	                         Search window
	                          <--------|
	Data                              PEC
	|----------------------------------|------------------------------------------|
	|                           XXXXXXXX                                          |
	|----------------------------------|------------------------------------------|
	                                   |
	Conveyor                           |
	|----------------------------------|------------------------------------------|
	|                      YYYYYYYY    |                                          |
	|                      YYYYYYYY    |                                          |
	|                      YYYYYYYY    |                                          |
	|----------------------------------|------------------------------------------|
	*)
	(* Data detected without PEC signal.*)
	            IF (#s_R_TRIG_PositiveDataFound.Q
	                AND NOT #sx_ParcelDetected)
	            THEN
	                #si_GINToWrite := 0;
	                // Double data detection loop.
	                FOR #si_i := #si_PositionToUpdate TO #si_PECPosition + (#si_SearchWindow * #si_Direction) BY #si_Direction DO
	                    // Data found in a search window.
	                    IF (#iqa_TrackingData[#si_i] > 0)
	                    THEN
	                        // First GIN found.
	                        IF (#si_GINToWrite = 0)
	                        THEN
	                            // Get the GIN if it's different than last updated GIN.
	                            IF #iqa_TrackingData[#si_i] <> #si_LastUpdatedGIN THEN
	                                #si_GINToWrite := #iqa_TrackingData[#si_i];
	                            END_IF;
	                            // If the first GIN was found, the scan loop conitues to check if there is no other data.
	                        ELSE
	                            // Next found data is different than the first one. Double data detected.
	                            IF (#iqa_TrackingData[#si_i] <> #si_GINToWrite)
	                            THEN
	                                #sx_DoubleDataFound := TRUE;
	                                // First found GIN is marked as a lost one and the GIN is stored in a FIFO register.
	                                IF ("DB_GIN".GIN[#si_GINToWrite].General.Lost = FALSE)
	                                THEN
	                                    "DB_GIN".GIN[#si_GINToWrite].General.Lost := TRUE;

	                                    "FC_Fifo"(ic_Mode := 'W',
	                                              qUDT_Status => #sUDT_LostGINFIFOStatus,
	                                              qx_Error => #sx_LostGINFIFOError,
	                                              qx_Warning => #sx_LostGINFIFOWarning,
	                                              iqv_Data := #si_GINToWrite,
	                                              iqUDT_FifoHeader := #iqUDT_FifoHeader,
	                                              iqv_DataBuffer := #iqa_FifoData);

	                                    // Update statistics
	                                    #ss_LostParcelsCounters.Total += 1;
	                                    #ss_LostParcelsCounters.DoubleData += 1;


	                                    ////////////////////

	                                    IF #si_GINToWrite >= 1000 THEN
	                                        #ss_LostValidParcelsCounters.Total += 1;
	                                        #ss_LostValidParcelsCounters.DoubleData += 1;
	                                    END_IF;

	                                    ////////////////
	                                END_IF;

	                                // Second found GIN is marked as a lost one and the GIN is stored in a FIFO register.
	                                IF ("DB_GIN".GIN[#iqa_TrackingData[#si_i]].General.Lost = FALSE)
	                                THEN
	                                    "DB_GIN".GIN[#iqa_TrackingData[#si_i]].General.Lost := TRUE;

	                                    "FC_Fifo"(ic_Mode := 'W',
	                                              qUDT_Status => #sUDT_LostGINFIFOStatus,
	                                              qx_Error => #sx_LostGINFIFOError,
	                                              qx_Warning => #sx_LostGINFIFOWarning,
	                                              iqv_Data := #iqa_TrackingData[#si_i],
	                                              iqUDT_FifoHeader := #iqUDT_FifoHeader,
	                                              iqv_DataBuffer := #iqa_FifoData);

	                                    // Update statistics
	                                    #ss_LostParcelsCounters.Total += 1;
	                                    #ss_LostParcelsCounters.DoubleData += 1;

	                                    ////////////////////

	                                    IF #iqa_TrackingData[#si_i] >= 1000 THEN
	                                        #ss_LostValidParcelsCounters.Total += 1;
	                                        #ss_LostValidParcelsCounters.DoubleData += 1;
	                                    END_IF;

	                                    ////////////////
	                                    //
	                                END_IF;
	                                // Stop search window scan in case of double data detection
	                                EXIT;
	                            END_IF;
	                        END_IF;
	                    END_IF;
	                END_FOR;

	                // Becasue the data was found as a first one, GIN is stored and the logic to wait for a parcel is enebaled.
	                // If the double data was found there is no need to wait for a parcel. Data has been marked as a lost one.
	                IF NOT #sx_DoubleDataFound
	                THEN
	                    #sx_ParcelWaitEnable := TRUE;
	                END_IF;

	                #sx_DoubleDataFound := FALSE;
	(*
	Data and PEC signal detected at the same time - perfect match

	                         Search window
	                          <--------|
	Data                              PEC
	|----------------------------------|------------------------------------------|
	|                           XXXXXXXX                                          |
	|----------------------------------|------------------------------------------|
	                                   |
	Conveyor                           |
	|----------------------------------|------------------------------------------|
	|                           XXXXXXXX                                          |
	|                           XXXXXXXX                                          |
	|                           XXXXXXXX                                          |
	|----------------------------------|------------------------------------------|

	or PEC signal found without data or with old ones

	                         Search window
	                          <--------|
	Data                              PEC
	|----------------------------------|------------------------------------------|
	|                    XXXXXXXX      |                                          |
	|----------------------------------|------------------------------------------|
	                                   |
	Conveyor                           |
	|----------------------------------|------------------------------------------|
	|                           XXXXXXXX                                          |
	|                           XXXXXXXX                                          |
	|                           XXXXXXXX                                          |
	|----------------------------------|------------------------------------------|
	*)
	(*Data and PEC signal detected at the same time (perfect match) or PEC signal found without data or with old ones.*)
	            ELSIF (#s_R_TRIG_ParcelFound.Q
	                AND (#s_R_TRIG_PositiveDataFound.Q
	                OR (#iqa_TrackingData[#si_PositionToUpdate] = 0
	                OR #iqa_TrackingData[#si_PositionToUpdate] = #si_LastUpdatedGIN)
	                AND NOT #sx_ParcelWaitEnable))
	            THEN
	                // If the PEC is set as a GIN generation point, skip data detection loop and go to GIN generator.
	                IF (#iUDT_PECUpdateConfiguration.GenerationPoint)
	                THEN
	                    #sx_GenerateGIN := TRUE;
	                    // If the the PEC isn't a generation point, data search loop is enabled.
	                ELSE
	                    #si_GINToWrite := 0;

	                    // Double data detection loop.
	                    FOR #si_i := #si_PositionToUpdate TO
	                        (#si_PECPosition + (#si_SearchWindow * #si_Direction)) BY #si_Direction DO

	                        // Data found in a search window.
	                        IF (#iqa_TrackingData[#si_i] > 0)
	                        THEN
	                            // First GIN found.
	                            IF (#si_GINToWrite = 0)
	                            THEN
	                                // Get the GIN if it's different than last updated GIN.
	                                IF #iqa_TrackingData[#si_i] <> #si_LastUpdatedGIN THEN
	                                    #si_GINToWrite := #iqa_TrackingData[#si_i];

	                                    // PEC/Data deviation acquisition
	                                    #"ss_PEC/DataDeviation".Last := DINT_TO_INT(#si_PECPosition - #si_i);
	                                    #"ss_PEC/DataDeviation".GIN := #si_GINToWrite;
	                                    #"ss_PEC/DataDeviation".Sum -= ABS(#"ss_PEC/DataDeviation".Last);
	                                    #"ss_PEC/DataDeviation".Nr += 1;
	                                    IF #"ss_PEC/DataDeviation".Last = 0 THEN
	                                        #"ss_PEC/DataDeviation".Type := 1;
	                                    ELSIF #"ss_PEC/DataDeviation".Last < 0 THEN
	                                        #"ss_PEC/DataDeviation".Type := 2;
	                                    END_IF;

	                                    // Parcel aligned statistics
	                                    IF (ABS(#"ss_PEC/DataDeviation".Last) > ABS(#si_Displacement - 1))
	                                    THEN
	                                        #ss_AlignedParcelsCounters.Total += 1;
	                                        #ss_AlignedParcelsCounters.PECNoData += 1;
	                                    END_IF;
	                                END_IF;
	                                // If the first GIN was found, the scan loop conitues to check if there is no other data.
	                            ELSE
	                                // Next found data is different than the first one. Double data detected.
	                                IF (#iqa_TrackingData[#si_i] <> #si_GINToWrite)
	                                THEN
	                                    // First found GIN is marked as a lost one and the GIN is stored in a FIFO register.
	                                    IF ("DB_GIN".GIN[#si_GINToWrite].General.Lost = FALSE)
	                                    THEN
	                                        "DB_GIN".GIN[#si_GINToWrite].General.Lost := TRUE;
	                                        "FC_Fifo"(ic_Mode := 'W',
	                                                  qUDT_Status => #sUDT_LostGINFIFOStatus,
	                                                  qx_Error => #sx_LostGINFIFOError,
	                                                  qx_Warning => #sx_LostGINFIFOWarning,
	                                                  iqv_Data := #si_GINToWrite,
	                                                  iqUDT_FifoHeader := #iqUDT_FifoHeader,
	                                                  iqv_DataBuffer := #iqa_FifoData);

	                                        // PEC/Data deviation acquisition
	                                        #"ss_PEC/DataDeviation".GIN := #si_GINToWrite;
	                                        #"ss_PEC/DataDeviation".Type := 4;

	                                        // Update statistics
	                                        #ss_LostParcelsCounters.Total += 1;
	                                        #ss_LostParcelsCounters.DoubleData += 1;

	                                        ////////////////////

	                                        IF #si_GINToWrite >= 1000 THEN
	                                            #ss_LostValidParcelsCounters.Total += 1;
	                                            #ss_LostValidParcelsCounters.DoubleData += 1;
	                                        END_IF;

	                                        ////////////////
	                                        //
	                                    END_IF;

	                                    // Second found GIN is marked as a lost one and the GIN is stored in a FIFO register.
	                                    IF ("DB_GIN".GIN[#iqa_TrackingData[#si_i]].General.Lost = FALSE)
	                                    THEN
	                                        "DB_GIN".GIN[#iqa_TrackingData[#si_i]].General.Lost := TRUE;
	                                        "FC_Fifo"(ic_Mode := 'W',
	                                                  qUDT_Status => #sUDT_LostGINFIFOStatus,
	                                                  qx_Error => #sx_LostGINFIFOError,
	                                                  qx_Warning => #sx_LostGINFIFOWarning,
	                                                  iqv_Data := #iqa_TrackingData[#si_i],
	                                                  iqUDT_FifoHeader := #iqUDT_FifoHeader,
	                                                  iqv_DataBuffer := #iqa_FifoData);

	                                        // Update statistics
	                                        #ss_LostParcelsCounters.Total += 1;
	                                        #ss_LostParcelsCounters.DoubleData += 1;

	                                        ////////////////////

	                                        IF #iqa_TrackingData[#si_i] >= 1000 THEN
	                                            #ss_LostValidParcelsCounters.Total += 1;
	                                            #ss_LostValidParcelsCounters.DoubleData += 1;
	                                        END_IF;

	                                        ////////////////
	                                        //
	                                    END_IF;
	                                    // Stop search window scan in case of double data detection
	                                    EXIT;
	                                END_IF;
	                            END_IF;
	                        END_IF;
	                    END_FOR;

	                    // GIN not found in a search window
	                    IF (#si_GINToWrite = 0)
	                    THEN
	                        #sx_GenerateGIN := TRUE;
	                        #si_UnknownParcelsCounters.DataNotFound += 1;
	                    END_IF;

	                    // Found GIN is a lost one - generate unknown GIN
	                    // Found GIN isn't lost or it's negative - don't do anything
	                    IF (#si_GINToWrite > 0)
	                    THEN
	                        IF ("DB_GIN".GIN[#si_GINToWrite].General.Lost)
	                        THEN
	                            #sx_GenerateGIN := TRUE;
	                            #si_UnknownParcelsCounters.LostParcelFound += 1;
	                        END_IF;
	                    END_IF;
	                END_IF;

	                (*Second parcel has been found during data update. Situation can occur when search window is too short
	                  and the data is shifted. In that case found GIN will be marked as a lost one and new unknown GIN will be
	                  generated. Negative GIN will be ignored.*)
	            ELSIF (#s_R_TRIG_ParcelFound.Q
	                AND (#iqa_TrackingData[#si_PositionToUpdate] <> 0
	                AND #iqa_TrackingData[#si_PositionToUpdate] <> #si_LastUpdatedGIN)
	                AND NOT #sx_ParcelWaitEnable)
	            THEN
	                IF (#iqa_TrackingData[#si_PositionToUpdate] > 0)
	                THEN
	                    IF ("DB_GIN".GIN[#iqa_TrackingData[#si_PositionToUpdate]].General.Lost = FALSE)
	                    THEN
	                        "DB_GIN".GIN[#iqa_TrackingData[#si_PositionToUpdate]].General.Lost := TRUE;
	                        "FC_Fifo"(ic_Mode := 'W',
	                                  qUDT_Status => #sUDT_LostGINFIFOStatus,
	                                  qx_Error => #sx_LostGINFIFOError,
	                                  qx_Warning => #sx_LostGINFIFOWarning,
	                                  iqv_Data := #iqa_TrackingData[#si_PositionToUpdate],
	                                  iqUDT_FifoHeader := #iqUDT_FifoHeader,
	                                  iqv_DataBuffer := #iqa_FifoData);

	                        // Update statistics
	                        #ss_LostParcelsCounters.Total += 1;
	                        #ss_LostParcelsCounters.DoubleData += 1;

	                        ////////////////////

	                        IF #iqa_TrackingData[#si_PositionToUpdate] >= 1000 THEN
	                            #ss_LostValidParcelsCounters.Total += 1;
	                            #ss_LostValidParcelsCounters.DoubleData += 1;
	                        END_IF;

	                        ////////////////
	                        //
	                    END_IF;
	                END_IF;

	                // Generate GIN
	                #sx_GenerateGIN := TRUE;
	                #si_UnknownParcelsCounters.LostParcelFound += 1;

	                (*Second data has been found during data update. Situation can occur when search window is too short
	                  and the data is shifted. In that case found GIN will be marked as a lost one.*)
	            ELSIF (#s_R_TRIG_PositiveDataFound.Q
	                AND #sx_ParcelDetected
	                AND #iqa_TrackingData[#si_PositionToUpdate] <> #si_GINToWrite)
	            THEN
	                // Mark GIN as a lost one
	                IF ("DB_GIN".GIN[#iqa_TrackingData[#si_PositionToUpdate]].General.Lost = FALSE)
	                THEN
	                    "DB_GIN".GIN[#iqa_TrackingData[#si_PositionToUpdate]].General.Lost := TRUE;
	                    "FC_Fifo"(ic_Mode := 'W',
	                              qUDT_Status => #sUDT_LostGINFIFOStatus,
	                              qx_Error => #sx_LostGINFIFOError,
	                              qx_Warning => #sx_LostGINFIFOWarning,
	                              iqv_Data := #iqa_TrackingData[#si_PositionToUpdate],
	                              iqUDT_FifoHeader := #iqUDT_FifoHeader,
	                              iqv_DataBuffer := #iqa_FifoData);

	                    // Update statistics
	                    #ss_LostParcelsCounters.Total += 1;
	                    #ss_LostParcelsCounters.DoubleData += 1;

	                    ////////////////////

	                    IF #iqa_TrackingData[#si_PositionToUpdate] >= 1000 THEN
	                        #ss_LostValidParcelsCounters.Total += 1;
	                        #ss_LostValidParcelsCounters.DoubleData += 1;
	                    END_IF;

	                    ////////////////
	                END_IF;
	            END_IF;

	        END_REGION

	        REGION 10.5 – GIN generator

	            (*Used to generate new GIN. If the PEC position is a generation point, the number is taken from an internal GIN range.
	              If it's not, then GIN is taken from a global unknown GIN range.*)

	            IF (#sx_GenerateGIN)
	            THEN
	                // Generation point.
	                IF (#iUDT_PECUpdateConfiguration.GenerationPoint)
	                THEN
	                    // Generate GIN from a valid GIN range.
	                    IF (#ss_ValidGINRange.GIN <= #ss_ValidGINRange.End)
	                    THEN
	                        #si_GINToWrite := #ss_ValidGINRange.GIN;
	                        #ss_ValidGINRange.GIN += 1;
	                    ELSE
	                        #si_GINToWrite := #ss_ValidGINRange.Start;
	                        #ss_ValidGINRange.GIN := #ss_ValidGINRange.Start + 1;
	                    END_IF;
	                    // Unknown GIN generator.
	                ELSE
	                    // Generate GIN from a unknown GIN range.
	                    IF (#iqUDT_UnknownGINRange.GIN <= #iqUDT_UnknownGINRange.End)
	                    THEN
	                        #si_GINToWrite := #iqUDT_UnknownGINRange.GIN;
	                        #iqUDT_UnknownGINRange.GIN += 1;
	                    ELSE
	                        #si_GINToWrite := #iqUDT_UnknownGINRange.Start;
	                        #iqUDT_UnknownGINRange.GIN := #iqUDT_UnknownGINRange.Start + 1;
	                    END_IF;

	                    // Unknwn parcels statistics.
	                    #si_UnknownParcelsCounters.Total += 1;
	                END_IF;

	                // Reset generte GIN command.
	                #sx_GenerateGIN := FALSE;

	                // GIN record is cleared with configured default GIN record while it's generated.
	                "DB_GIN".GIN[#si_GINToWrite] := "DB_GINDefault".GIN[#iUDT_PECUpdateConfiguration.DefaultGIN];
	            END_IF;

	            #qi_GINwrite := #si_GINToWrite;

	        END_REGION


	        REGION 10.6 – PEC position data update

	            (*While parcel is detected, calculated GIN is written into the PEC position record.
	              If not, then the record is cleared with 0. Negative GIN is ignored or deleted, depending on configuration.*)

	            IF (#sx_ParcelDetected)
	            THEN

	                "FC_WriteGIN"(ii_GIN := #si_GINToWrite,
	                              ii_PositionToWrite := #si_PositionToUpdate,
	                              ii_NumberOfPositions := 1,
	                              ix_Direction := TRUE,
	                              iqa_TrackingData := #iqa_TrackingData);

	            ELSE
	                IF (#iqa_TrackingData[#si_PositionToUpdate] > 0
	                    OR #iUDT_PECUpdateConfiguration.NegativeGINDelete)
	                THEN

	                    "FC_WriteGIN"(ii_GIN := #ci_ZeroGIN,
	                                  ii_PositionToWrite := #si_PositionToUpdate,
	                                  ii_NumberOfPositions := 1,
	                                  ix_Direction := TRUE,
	                                  iqa_TrackingData := #iqa_TrackingData);

	                END_IF;
	            END_IF;

	        END_REGION

	        REGION 10.7 – Parcel waiting logic

	            (*Parcel waiting logic is used to wait for the photoeye signal for a search window distance.*)
	            IF (#sx_ParcelWaitEnable)
	            THEN
	                // Counting parcel wait distance depending on conveyor running direction if not detected.
	                IF (NOT #sx_ParcelDetected)
	                THEN
	                    IF (#si_Direction = 1)
	                    THEN
	                        #si_ParcelWaitDistance += 1;

	                    ELSE
	                        #si_ParcelWaitDistance -= ABS(#si_Displacement);   //1;
	                    END_IF;

	                    // Parcel detected - stop waiting, use found GIN to update.
	                ELSE
	                    // PEC/Data deviation acquisition
	                    #"ss_PEC/DataDeviation".Type := 3;
	                    #"ss_PEC/DataDeviation".Last := #si_ParcelWaitDistance;
	                    #"ss_PEC/DataDeviation".GIN := #si_GINToWrite;
	                    #"ss_PEC/DataDeviation".Sum += ABS(#"ss_PEC/DataDeviation".Last);
	                    #"ss_PEC/DataDeviation".Nr += 1;


	                    // Parcel aligned statistics
	                    IF (#"ss_PEC/DataDeviation".Last > ABS(#si_Displacement - 1))
	                    THEN
	                        #ss_AlignedParcelsCounters.Total += 1;
	                        #ss_AlignedParcelsCounters.DataNoPEC += 1;
	                    END_IF;

	                    // Parcel waiting logic reset.
	                    #sx_ParcelWaitEnable := FALSE;
	                    #si_ParcelWaitDistance := 0;
	                END_IF;
	            END_IF;

	            // Parcel not found in a search window - stop waiting, mark found GIN as a lost one.
	            IF (ABS(#si_ParcelWaitDistance) = #si_SearchWindow)
	                AND (#si_GINToWrite > 0)
	            THEN
	                // Parcel lost
	                IF "DB_GIN".GIN[#si_GINToWrite].General.Lost = FALSE THEN
	                    "DB_GIN".GIN[#si_GINToWrite].General.Lost := TRUE;
	                    "FC_Fifo"(ic_Mode := 'W',
	                              qUDT_Status => #sUDT_LostGINFIFOStatus,
	                              qx_Error => #sx_LostGINFIFOError,
	                              qx_Warning => #sx_LostGINFIFOWarning,
	                              iqv_Data := #si_GINToWrite,
	                              iqUDT_FifoHeader := #iqUDT_FifoHeader,
	                              iqv_DataBuffer := #iqa_FifoData);

	                    // PEC/Data deviation acquisition
	                    #"ss_PEC/DataDeviation".Type := 5;
	                    #"ss_PEC/DataDeviation".Last := #si_ParcelWaitDistance;
	                    #"ss_PEC/DataDeviation".GIN := #si_GINToWrite;
	                    #"ss_PEC/DataDeviation".Sum += ABS(#"ss_PEC/DataDeviation".Last);
	                    #"ss_PEC/DataDeviation".Nr += 1;

	                    // Parcel waiting logic reset.
	                    #si_ParcelWaitDistance := 0;
	                    #sx_ParcelWaitEnable := FALSE;

	                    // Lost parcels ina  row counter.
	                    #si_LostParcelsInARow += 1;

	                    // Update statistics.
	                    #ss_LostParcelsCounters.Total += 1;
	                    #ss_LostParcelsCounters.ParcelNotFound += 1;

	                    ////////////////////

	                    IF #si_GINToWrite >= 1000 THEN
	                        #ss_LostValidParcelsCounters.Total += 1;
	                        #ss_LostValidParcelsCounters.ParcelNotFound += 1;
	                    END_IF;

	                    ////////////////
	                    //
	                END_IF;

	            END_IF;

	            // Reset monitoring in case of going backwards.
	            IF (#si_ParcelWaitDistance = 0
	                AND NOT #sx_ParcelDetected
	                AND #sx_InvalidDirection)
	            THEN
	                #sx_ParcelWaitEnable := FALSE;
	            END_IF;

	            #sx_InvalidDirection := ((#si_Direction = 1
	            AND #si_ParcelWaitDistance < 0)
	            OR (#si_Direction = -1
	            AND #si_ParcelWaitDistance > 0));

	        END_REGION

	        REGION 10.8 – Last updated GIN

	            (*Last updated GIN to avoid processing the same data.*)
	            IF (#s_R_TRIG_DataFound.Q)
	            THEN
	                #si_LastUpdatedGIN := #iqa_TrackingData[#si_PositionToUpdate];
	            END_IF;

	        END_REGION

	        REGION 10.8 – Update displacement

	            #si_Displacement := #si_Displacement - #si_Direction;

	        END_REGION

	    END_WHILE;

	END_REGION

	REGION 11 – Length measurement



	    (*Length and gap measurements can be enabled via PEC update configuration*)
	    #sFB_LengthMeasurement(ii_PECPosition := #si_PECPosition,
	                           ii_Displacement := #iqUDT_ConveyorInterface.Displacement,
	                           ix_LengthMeasurementEnable := #iUDT_PECUpdateConfiguration.ParcelLengthMeasurement OR #sx_LengthMeasurementEnable,
	                           ix_GapMeasurementEnable := #iUDT_PECUpdateConfiguration.GapLengthMeasurement,
	                           iqa_TrackingData := #iqa_TrackingData);

	    IF #iqa_TrackingData[#si_PECPosition] > 0
	        AND #iqa_TrackingData[#si_PECPosition] >= #iqUDT_UnknownGINRange.Start
	        AND #iqa_TrackingData[#si_PECPosition] <= #iqUDT_UnknownGINRange.End
	    THEN

	        #sx_LengthMeasurementEnable := "DB_GIN".GIN[#iqa_TrackingData[#si_PECPosition]].General.Length = 0;
	    ELSE

	        #sx_LengthMeasurementEnable := FALSE;

	    END_IF;

	END_REGION

	REGION 12 – Teaching done

	    // Average slip calculation
	    #si_AverageSlip := #"ss_PEC/DataDeviation".Sum / #"ss_PEC/DataDeviation".Nr;
	    #si_CalculatedLengthCorrection := DINT_TO_INT(#iUDT_ConveyorCommonConfiguration.LengthCorrection) + #si_AverageSlip * 10;
	    IF (#sx_TeachingMode                                                                                                            // Teaching mode enabled
	        AND #si_NumberOfTeachedParcels = #iUDT_PECUpdateConfiguration.NrOfTeachParcels)                                                 // Number of teaching parcels equal to the preset one                                                                                                                                                              // Teaching mode enabled ("sx_TeachMode")
	    THEN

	        #si_CalculatedLengthCorrection := DINT_TO_INT(#iUDT_ConveyorCommonConfiguration.LengthCorrection) + #si_AverageSlip * 10;
	        #sx_TeachingMode := FALSE;
	        #si_NumberOfTeachedParcels := 0;

	    END_IF;

	END_REGION

	REGION 13 – Performance

	    (*Performnce is a percentage ratio between number of lost parcels and total number of data, used to monitor data update efficiency.*)

	    IF (#sdi_TotalNumberOfData >= #ss_LostParcelsCounters.Total
	        AND #sdi_TotalNumberOfData > 0)
	    THEN
	        #slr_Performance := 100.0 - INT_TO_LREAL(#ss_LostParcelsCounters.Total) / #sdi_TotalNumberOfData * 100.0;
	    END_IF;

	    // Warning is generated if performance drops below 80%.
	    #qUDT_Status.LowPerformance := #slr_Performance < 80;

	END_REGION

	REGION 14 – Reset statistics

	    // Statistics are reset if reset signal is given.
	    IF #iqUDT_ConveyorInterface.ResetStatistics
	    THEN
	        #sdi_TotalNumberOfParcels := 0;
	        #ss_AlignedParcelsCounters.Total := 0;
	        #ss_AlignedParcelsCounters.PECNoData := 0;
	        #ss_AlignedParcelsCounters.DataNoPEC := 0;
	        #ss_LostParcelsCounters.Total := 0;
	        #ss_LostParcelsCounters.DoubleData := 0;
	        #ss_LostParcelsCounters.ParcelNotFound := 0;
	        #ss_LostValidParcelsCounters.Total := 0;
	        #ss_LostValidParcelsCounters.DoubleData := 0;
	        #ss_LostValidParcelsCounters.ParcelNotFound := 0;
	        #sdi_TotalNumberOfData := 0;
	        #si_UnknownParcelsCounters.Total := 0;
	        #si_UnknownParcelsCounters.LostParcelFound := 0;
	        #si_UnknownParcelsCounters.DataNotFound := 0;
	        #"ss_PEC/DataDeviation".Sum := 0;
	        #"ss_PEC/DataDeviation".Nr := 0;
	        #slr_Performance := 100;

	    END_IF;

	END_REGION

	REGION 15 – Too many lost parcels error

	    (*Error is generated if too many parcels will is marked as a lost one in a row*)
	    IF (#si_LostParcelsInARow >= #iUDT_PECUpdateConfiguration.MaxLost)
	    THEN
	        #qUDT_Status.TooManyLost := TRUE;
	    END_IF;

	END_REGION

	REGION 16 – Statistics

	    // Too many lost
	    #s_R_TRIG_TooManyLost(CLK := #qUDT_Status.TooManyLost);
	    IF #qUDT_Status.TooManyLost
	        OR #iqUDT_ConveyorInterface.ResetStatistics
	    THEN
	        "FC_Statistics"(ix_Reset := #iqUDT_ConveyorInterface.ResetStatistics,
	                        ix_Activate := #qUDT_Status.TooManyLost,
	                        ix_RTrigActivate := #s_R_TRIG_TooManyLost.Q,
	                        iqUDT_Statistics := #iqUDT_Statistics.TooManyLost);
	    END_IF;

	    // Total number of parcels
	    #iqUDT_Statistics.TotalNrOfParcels := #sdi_TotalNumberOfParcels;

	END_REGION

	REGION 17 – Internal tracking warning and error

	    // Internal tracking warning
	    IF (#qUDT_Status.LowPerformance
	        OR #sx_LostGINFIFOWarning)
	    THEN
	        #iqUDT_ConveyorInterface.InternalWarningTracking := TRUE;
	    END_IF;

	    // Internal tracking error
	    IF #qUDT_Status.TooManyLost
	    THEN
	        #iqUDT_ConveyorInterface.InternalErrorTracking := TRUE;
	    END_IF;

	    // Configuration error
	    IF (#sx_InvalidDisplacement
	        OR #sx_InvalidGINRange
	        OR #sx_InvalidSearchWindow)
	    THEN
	        #iqUDT_ConveyorInterface.ConfigurationError := TRUE;
	    END_IF;

	END_REGION
END_FUNCTION_BLOCK

FUNCTION_BLOCK "FB_CaljanV2"
TITLE = FB_Unloader
{ S7_Optimized_Access := 'TRUE' }
AUTHOR : MHSE
FAMILY : Equimpent
VERSION : 1.2
// ATTRIBUTES
// AUTO_NUMBER = True
// BLOCK_NUMBER = 201
// END_ATTRIBUTES
//Function block to control unloader.
   VAR_INPUT
      iUDT_CaljanConfiguration { ExternalAccessible := 'False'; ExternalVisible := 'False'; ExternalWritable := 'False'} : "UDT_CaljanConfigurationV2";   // Caljan configuration structure
      iUDT_CaljanReceive { ExternalAccessible := 'False'; ExternalVisible := 'False'; ExternalWritable := 'False'} : "UDT_CaljanReceiveV2";   // Caljan receive structure
      ix_SafetyReset { ExternalAccessible := 'False'; ExternalVisible := 'False'; ExternalWritable := 'False'} : Bool;   // Safety reset
      ix_SafetyOk { ExternalAccessible := 'False'; ExternalVisible := 'False'; ExternalWritable := 'False'} : Bool;   // TRUE when Safety Circuit of the Conveyor is healthy
      ix_24vOk { ExternalAccessible := 'False'; ExternalVisible := 'False'; ExternalWritable := 'False'} : Bool;   // TRUE when 24VDC is healthy
      ix_400vOk { ExternalAccessible := 'False'; ExternalVisible := 'False'; ExternalWritable := 'False'} : Bool;   // TRUE when 400VAC is healthy
      ix_HardwareOK { ExternalAccessible := 'False'; ExternalVisible := 'False'; ExternalWritable := 'False'} : Bool;   // TRUE when the PN node(s) are ok
      ix_ExternalRequestDieBack { ExternalAccessible := 'False'; ExternalVisible := 'False'; ExternalWritable := 'False'} : Bool;   // External request die back
      ix_ExternalRequestHold { ExternalAccessible := 'False'; ExternalVisible := 'False'; ExternalWritable := 'False'} : Bool;   // External request hold
      ix_ExternalRunReverse { ExternalAccessible := 'False'; ExternalVisible := 'False'; ExternalWritable := 'False'} : Bool;   // External request only for unloder mode - TRUE when conveyor should run in reverse direction
      ix_ResetEnergySave { ExternalAccessible := 'False'; ExternalVisible := 'False'; ExternalWritable := 'False'} : Bool;   // Reset energy save mode timer
      ix_SimulationModeActive { ExternalAccessible := 'False'; ExternalVisible := 'False'; ExternalWritable := 'False'} : Bool;   // TRUE when simulation mode is active
      ix_CaljanMode { ExternalAccessible := 'False'; ExternalVisible := 'False'; ExternalWritable := 'False'} : Int;   // Choosing device 1=loader, 2=unloader
      ix_BufferPEC { ExternalAccessible := 'False'; ExternalVisible := 'False'; ExternalWritable := 'False'} : Bool;   // Buufer PEC
   END_VAR

   VAR_OUTPUT
      qUDT_HMIStatus { ExternalAccessible := 'False'; ExternalVisible := 'False'; ExternalWritable := 'False'} : "UDT_CaljanStatusV2";   // HMI status structure
      qUDT_Status { ExternalAccessible := 'False'; ExternalVisible := 'False'; ExternalWritable := 'False'} : "UDT_CommonStatus";   // Common status structure
      qUDT_CaljanSend { ExternalAccessible := 'False'; ExternalVisible := 'False'; ExternalWritable := 'False'} : "UDT_CaljanSendV2";   // Caljan send structure
   END_VAR

   VAR_IN_OUT
      iqUDT_EquipmentControl : "UDT_EquipmentControl";   // Equipment control structure
      iqUDT_CaljanCommand : "UDT_CaljanCommand";   // Caljan HMI control
      iqUDT_ConveyorInterface : "UDT_ConveyorInterface";   // Interface structure
      iqUDT_HandShake : "UDT_ConveyorHandshake";   // Handshake structure
      iqUDT_HandShakeUp : "UDT_ConveyorHandshake";   // Upstream handshake structure
      iqUDT_Statistics : "UDT_CaljanStatisticsV2";   // Statistics structure
   END_VAR

   VAR
      s_FB_ResetPulseTimer { ExternalAccessible := 'False'; ExternalVisible := 'False'; ExternalWritable := 'False'; S7_SetPoint := 'False'} : "FB_TimerOnOffDelay";   // Timer on/off delay for reset pulse
      s_FB_CascadeModeTimer { ExternalAccessible := 'False'; ExternalVisible := 'False'; ExternalWritable := 'False'; S7_SetPoint := 'False'} : "FB_TimerOnOffDelay";   // Timer on/off delay for cascade mode
      s_FB_TimerOnOffDelayCheck24V { ExternalAccessible := 'False'; ExternalVisible := 'False'; ExternalWritable := 'False'; S7_SetPoint := 'False'} : "FB_TimerOnOffDelay";   // Timer on/off delay to allow startup before fault is generated
      s_FB_TimerOnOffDelayCheck400V { ExternalAccessible := 'False'; ExternalVisible := 'False'; ExternalWritable := 'False'; S7_SetPoint := 'False'} : "FB_TimerOnOffDelay";   // Timer on/off delay to allow startup before fault is generated
      s_UDT_CommonStatus { ExternalAccessible := 'False'; ExternalVisible := 'False'; ExternalWritable := 'False'; S7_SetPoint := 'False'} : "UDT_CommonStatus";   // Common status structure
      s_UDT_CommonStatusOld { ExternalAccessible := 'False'; ExternalVisible := 'False'; ExternalWritable := 'False'; S7_SetPoint := 'False'} : "UDT_CommonStatus";   // Auxiliary status structure
      s_UDT_HMIStatus { ExternalAccessible := 'False'; ExternalVisible := 'False'; ExternalWritable := 'False'; S7_SetPoint := 'False'} : "UDT_CaljanStatusV2";   // HMI status structure
      s_UDT_PNDevice { ExternalAccessible := 'False'; ExternalVisible := 'False'; ExternalWritable := 'False'; S7_SetPoint := 'False'} : "UDT_PNDevice";   // PN device info structure
      sa_PNPortsStatus { ExternalAccessible := 'False'; ExternalVisible := 'False'; ExternalWritable := 'False'} : Array[1..8] of Bool;   // TRUE when specific port has an error
      R_TRIG_EnergySave {InstructionName := 'R_TRIG'; LibVersion := '1.0'; ExternalAccessible := 'False'; ExternalVisible := 'False'; ExternalWritable := 'False'; S7_SetPoint := 'False'} : R_TRIG;   // Rising edge for energy save
      R_TRIG_ConveyorUp {InstructionName := 'R_TRIG'; LibVersion := '1.0'; ExternalAccessible := 'False'; ExternalVisible := 'False'; ExternalWritable := 'False'; S7_SetPoint := 'False'} : R_TRIG;   // Rising edge of automatic active
      R_TRIG_ConveyorDown {InstructionName := 'R_TRIG'; LibVersion := '1.0'; ExternalAccessible := 'False'; ExternalVisible := 'False'; ExternalWritable := 'False'; S7_SetPoint := 'False'} : R_TRIG;   // Rising edge of automatic not active
      R_TRIG_NotHealthy {InstructionName := 'R_TRIG'; LibVersion := '1.0'; ExternalAccessible := 'False'; ExternalVisible := 'False'; ExternalWritable := 'False'; S7_SetPoint := 'False'} : R_TRIG;   // Rising edge trigger if extendable not healthy
      R_TRIG_SafetyOk {InstructionName := 'R_TRIG'; LibVersion := '1.0'; ExternalAccessible := 'False'; ExternalVisible := 'False'; ExternalWritable := 'False'; S7_SetPoint := 'False'} : R_TRIG;   // Rising edge trigger safety is ok
      s_R_TRIG_PNSlaveError {InstructionName := 'R_TRIG'; LibVersion := '1.0'; ExternalAccessible := 'False'; ExternalVisible := 'False'; ExternalWritable := 'False'; S7_SetPoint := 'False'} : R_TRIG;   // Rising edge for PN error
      s_R_TRIG_PNSlaveNotOnline {InstructionName := 'R_TRIG'; LibVersion := '1.0'; ExternalAccessible := 'False'; ExternalVisible := 'False'; ExternalWritable := 'False'; S7_SetPoint := 'False'} : R_TRIG;   // Rising edge for PN not online
      s_R_TRIG_ResetEnergySaveRunMode {InstructionName := 'R_TRIG'; LibVersion := '1.0'; ExternalAccessible := 'False'; ExternalVisible := 'False'; ExternalWritable := 'False'; S7_SetPoint := 'False'} : R_TRIG;   // Rising edge trigger reset energy save mode
      s_R_TRIG_ResetEnergySaveBufferMode {InstructionName := 'R_TRIG'; LibVersion := '1.0'; ExternalAccessible := 'False'; ExternalVisible := 'False'; ExternalWritable := 'False'; S7_SetPoint := 'False'} : R_TRIG;   // Rising edge trigger reset energy save mode
      s_R_TRIG_ResetEnergySaveActive {InstructionName := 'R_TRIG'; LibVersion := '1.0'; ExternalAccessible := 'False'; ExternalVisible := 'False'; ExternalWritable := 'False'; S7_SetPoint := 'False'} : R_TRIG;   // Rising edge trigger reset energy save mode
   END_VAR
   VAR RETAIN
      sdi_EnergySave { ExternalAccessible := 'False'; ExternalVisible := 'False'; ExternalWritable := 'False'} : DInt;   // Energy save displacement
   END_VAR
   VAR
      sx_Disabled { ExternalAccessible := 'False'; ExternalVisible := 'False'; ExternalWritable := 'False'} : Bool;   // Operation is enabled
      sx_Ready { ExternalAccessible := 'False'; ExternalVisible := 'False'; ExternalWritable := 'False'} : Bool;   // Conveyor Ready to operate in Forward mode
      sx_EnergySaveActive { ExternalAccessible := 'False'; ExternalVisible := 'False'; ExternalWritable := 'False'} : Bool;   // Active energy save mode
      sx_AutomaticActive { ExternalAccessible := 'False'; ExternalVisible := 'False'; ExternalWritable := 'False'} : Bool;   // Forward active
      sx_CascadeStartUp { ExternalAccessible := 'False'; ExternalVisible := 'False'; ExternalWritable := 'False'} : Bool;   // Cascade startup auxiliary bit
      sx_24VOk { ExternalAccessible := 'False'; ExternalVisible := 'False'; ExternalWritable := 'False'} : Bool;   // 24V ok
      sx_400VOk { ExternalAccessible := 'False'; ExternalVisible := 'False'; ExternalWritable := 'False'} : Bool;   // 400V ok
   END_VAR

   VAR CONSTANT
      ci_NumberOfProfinetPorts : Int := 2;   // Number of Profinet ports in device
      ci_PowerSupplyDelayTime : UInt := 4000;   // Power supply delay time
   END_VAR


BEGIN
	(*
	----------------------------------------------------------------------------------------
	|                                                                                      |
	|  Copyright  2023             FORTNA Europe BV                                        |
	|  All Rights Reserved         Netherlands                                             |
	|                                                                                      |
	----------------------------------------------------------------------------------------

	Version history:
	Date        | Version   | Author       | Remark
	----------------------------------------------------------------------------------------
	07/03/2023  | 1.0       | S. Nikodem   | Release TIA 17 | DHL Munich 2023
	20/12/2023  | 1.1       | M. Diebel    | Update
	20/12/2023  | 1.2       | L.Klar       | Energy save mode added
	05/02/20234 | 1.3       | P.Gryszczyk  | Added HardwareOk to Profinet faults reset
	05/02/20234 | 1.4       | L.Klar       | Added dieback condition to unload function
	07/02/20234 | 1.5       | L.Klar       | Buffer mode corrected
	09/02/2024  | 1.6       | P.Gryszczyk  | Changed logic for BufferPEC when using Caljan sensor
	*)

	REGION 1 - Get Device Profinet information

	    "FC_GetDevicePN"(is_PNDeviceName := #iUDT_CaljanConfiguration.PNDeviceName,
	                     ix_SimulationModeActive := #ix_SimulationModeActive,
	                     iqUDT_PND := #s_UDT_PNDevice);

	    "FC_GetPNPortStatus"(ii_NumberOfPorts := #ci_NumberOfProfinetPorts,
	                         iUDT_DevicePNInfo := #s_UDT_PNDevice,
	                         qa_PortFault => #sa_PNPortsStatus);

	END_REGION

	REGION 2 - Initial

	    REGION 2.1 - First PLC cycle

	        IF "DB_Memory".FirstScan
	        THEN
	            #sx_AutomaticActive := FALSE;
	            #iqUDT_HandShakeUp.RTR := FALSE;
	            #iqUDT_HandShakeUp.CascadeStartUp := FALSE;
	            #sx_Disabled := FALSE;
	        END_IF;

	    END_REGION

	    REGION 2.2 - Triggers

	        // Rising edge trigger energy save
	        #R_TRIG_EnergySave(CLK := #s_UDT_CommonStatus.EnergySave);

	        // Rising edge extendable up
	        #R_TRIG_ConveyorUp(CLK := #sx_AutomaticActive AND #sx_Ready);

	        // Rising edge extendable down
	        #R_TRIG_ConveyorDown(CLK := #sx_AutomaticActive AND NOT #sx_Ready);

	        // Rising edge extendable not healthy
	        #R_TRIG_NotHealthy(CLK := #s_UDT_HMIStatus.Specific.NotHealthy);

	        // Rising edge for Profinet error
	        #s_R_TRIG_PNSlaveError(CLK := #s_UDT_HMIStatus.Specific.PNSlaveError);

	        // Rising edge for Profinet not online
	        #s_R_TRIG_PNSlaveNotOnline(CLK := #s_UDT_HMIStatus.Specific.PNSlaveNotOnline);

	        // Rising edge for reset energy save mode

	        #s_R_TRIG_ResetEnergySaveRunMode(CLK := #iUDT_CaljanReceive.RunModeActivated);
	        #s_R_TRIG_ResetEnergySaveBufferMode(CLK := #iUDT_CaljanReceive.StoreModeActivated);
	        #s_R_TRIG_ResetEnergySaveActive(CLK := #sx_EnergySaveActive);


	    END_REGION

	    REGION 2.3 - HMI button Disable operation

	        // Copy HMI command to static memory
	        #sx_Disabled := #iqUDT_CaljanCommand.Disable;

	        // Copy status to HMI
	        #s_UDT_HMIStatus.Specific.Disabled := #sx_Disabled;

	    END_REGION

	    REGION 2.6 - Timers

	        // Hardware will only be available after the delay, so the device has time for the initialisation
	        #s_FB_TimerOnOffDelayCheck24V(iudi_OnDelayTime := #ci_PowerSupplyDelayTime,
	                                      ix_SignalToDelay := #ix_24vOk,
	                                      qx_DelayedSignal => #sx_24VOk);

	        #s_FB_TimerOnOffDelayCheck400V(iudi_OnDelayTime := #ci_PowerSupplyDelayTime,
	                                       ix_SignalToDelay := #ix_400vOk,
	                                       qx_DelayedSignal => #sx_400VOk);

	    END_REGION

	END_REGION

	REGION 3 - Reset Profinet errors

	    IF #iqUDT_EquipmentControl.Command.Reset OR (NOT #ix_HardwareOK AND #s_UDT_HMIStatus.Specific.PNSlaveNotOnline) THEN

	        #s_UDT_HMIStatus.Specific.PNSlaveNotOnline := FALSE;
	        #s_UDT_HMIStatus.Specific.PNSlaveError := FALSE;
	        #s_UDT_HMIStatus.Specific.PNSlaveWarning := FALSE;
	    END_IF;

	END_REGION

	REGION 4 - Errors

	    // Check if PN device is online
	    IF NOT "DB_ProfinetDiagnostic".ProfinetNetworks[#s_UDT_PNDevice.PNNetworknumber].DeviceStatus[#s_UDT_PNDevice.PNDeviceNumber].DeviceState.Exist
	        AND NOT #ix_SimulationModeActive
	        AND #sx_24VOk
	        AND #ix_HardwareOK
	    THEN
	        #s_UDT_HMIStatus.Specific.PNSlaveNotOnline := TRUE;

	    END_IF;

	    // Check if PN ports are healthy
	    IF #sa_PNPortsStatus[1] XOR #sa_PNPortsStatus[2] THEN
	        #s_UDT_HMIStatus.Specific.PNSlaveWarning := TRUE;
	    END_IF;

	    // Check if PN device has an error
	    IF "DB_ProfinetDiagnostic".ProfinetNetworks[#s_UDT_PNDevice.PNNetworknumber].DeviceStatus[#s_UDT_PNDevice.PNDeviceNumber].DeviceState.Error
	        AND NOT #ix_SimulationModeActive
	        AND #sx_24VOk
	        AND NOT #s_UDT_HMIStatus.Specific.PNSlaveWarning
	        AND #ix_HardwareOK
	    THEN
	        #s_UDT_HMIStatus.Specific.PNSlaveError := TRUE;
	    END_IF;

	    // Not healthy
	    #s_UDT_HMIStatus.Specific.NotHealthy := NOT #iUDT_CaljanReceive.Healthy
	    AND #sx_400VOk
	    AND #sx_24VOk
	    AND #ix_HardwareOK
	    AND #ix_SafetyOk;

	    // Common Error
	    #s_UDT_CommonStatus.Error := NOT #sx_24VOk
	    OR NOT #sx_400VOk
	    OR NOT #ix_HardwareOK
	    OR NOT #ix_SafetyOk
	    OR #s_UDT_HMIStatus.Specific.PEC_EoS.Jam
	    OR #s_UDT_HMIStatus.Specific.NotHealthy;


	END_REGION

	REGION 5 - Speed

	    #iqUDT_ConveyorInterface.ActualSpeed := #iUDT_CaljanReceive.ActualSpeed;

	END_REGION

	REGION 6 - Check conditions to set caljan ready

	    #sx_Ready := NOT #s_UDT_CommonStatus.Error;

	END_REGION

	REGION 7 - Stop caljan

	    IF NOT #iqUDT_EquipmentControl.Command.AutomaticOn
	        OR #s_UDT_CommonStatus.Error
	    THEN
	        #sx_AutomaticActive := FALSE;
	        #qUDT_CaljanSend.AllowLoading := FALSE;
	        #qUDT_CaljanSend.AllowUnloading := FALSE;
	        #iqUDT_HandShakeUp.RTR := FALSE;
	        #iqUDT_HandShakeUp.CascadeStartUp := FALSE;
	    END_IF;

	END_REGION

	REGION 8 - Start automatic mode

	    // If start (one shot) is received from system, this is memorised until started in cascade. Later the unloader is started
	    IF #iqUDT_EquipmentControl.Command.Start
	        AND #sx_Ready
	    THEN
	        #sx_AutomaticActive := TRUE;
	    END_IF;

	    //Timer to cascade mode
	    #s_FB_CascadeModeTimer(iudi_OnDelayTime := #iUDT_CaljanConfiguration.CascadeTimeOnDelay,
	                           ix_SignalToDelay := #sx_AutomaticActive,
	                           ix_Enable := #sx_Ready,
	                           qx_DelayedSignal => #sx_CascadeStartUp);

	    #iqUDT_HandShakeUp.CascadeStartUp := #sx_CascadeStartUp;

	    //Automatic mode active
	    #qUDT_CaljanSend.Enable := #sx_AutomaticActive AND NOT #s_R_TRIG_ResetEnergySaveActive.Q;

	END_REGION

	REGION 9 - Automatic mode active

	    REGION 9.1 - Operation

	        (* *******LOADER ******** *)
	        IF #ix_CaljanMode = 1 THEN

	            // Release loading
	            #qUDT_CaljanSend.AllowLoading := #sx_AutomaticActive
	            AND #sx_Ready
	            AND NOT #sx_Disabled
	            AND NOT #ix_ExternalRequestHold
	            AND NOT #sx_EnergySaveActive
	            AND (#iUDT_CaljanReceive.RunModeActivated OR #iUDT_CaljanReceive.StoreModeActivated);

	            #iqUDT_HandShakeUp.RTR := #qUDT_CaljanSend.AllowLoading AND ABS(#iUDT_CaljanReceive.ActualSpeed) > 400;

	        END_IF;

	        (* *******UNLOADER ******** *)
	        IF #ix_CaljanMode = 2
	        THEN

	            // Release unloading
	            #qUDT_CaljanSend.AllowUnloading := #sx_AutomaticActive
	            AND #sx_Ready
	            AND (#iqUDT_HandShake.RTR OR #iUDT_CaljanReceive.PECUnloader)
	            AND NOT #sx_Disabled
	            AND NOT #ix_ExternalRequestHold
	            AND NOT #sx_EnergySaveActive
	            AND NOT #ix_ExternalRunReverse;

	        END_IF;

	    END_REGION

	    REGION 9.2 - Energy save

	        IF #iUDT_CaljanConfiguration.Energy THEN


	            IF #sdi_EnergySave >= #iUDT_CaljanConfiguration.EnergySaveLenght        // Compare energy save counter with configured lenght
	            THEN
	                #sx_EnergySaveActive := TRUE;                                           // Set energy save active true
	            END_IF;

	            (* *******LOADER ******** *)
	            // Reset
	            IF (#ix_CaljanMode = 1
	                AND (NOT #iUDT_CaljanReceive.PECUnloader
	                OR NOT #iUDT_CaljanReceive.PECLoader)
	                AND NOT #sx_EnergySaveActive)
	                OR #ix_ResetEnergySave
	                OR #iqUDT_HandShakeUp.RTS
	                OR #iqUDT_HandShakeUp.ResetEnergySave
	                OR NOT #iqUDT_EquipmentControl.Command.AutomaticOn
	                OR #s_R_TRIG_ResetEnergySaveBufferMode.Q
	                OR #s_R_TRIG_ResetEnergySaveRunMode.Q
	            THEN
	                #sx_EnergySaveActive := FALSE;
	                #sdi_EnergySave := 0;

	                (* *******UNLOADER ******** *)
	            ELSIF (#ix_CaljanMode = 2
	                AND (NOT #iUDT_CaljanReceive.PECUnloader
	                OR NOT #iUDT_CaljanReceive.PECLoader)
	                AND NOT #sx_EnergySaveActive)
	                OR #ix_ResetEnergySave
	                OR #s_R_TRIG_ResetEnergySaveBufferMode.Q
	                OR #s_R_TRIG_ResetEnergySaveRunMode.Q
	            THEN
	                #sx_EnergySaveActive := FALSE;
	                #sdi_EnergySave := 0;

	            ELSE

	                #sdi_EnergySave += ABS(#iqUDT_ConveyorInterface.Displacement);

	            END_IF;
	        ELSE

	            #sx_EnergySaveActive := FALSE;
	            #sdi_EnergySave := 0;

	        END_IF;

	        IF #sx_AutomaticActive
	        THEN
	            #iqUDT_HandShake.ResetEnergySave := NOT #iUDT_CaljanReceive.PECUnloader AND NOT #sx_EnergySaveActive;
	        END_IF;

	    END_REGION

	    REGION 9.3 Buffer PEC

	        IF #iUDT_CaljanConfiguration.BufferPEC THEN

	            #qUDT_CaljanSend.BufferPEC := #ix_BufferPEC;

	        ELSE
	            //When in store mode we using Caljan's Unloader PEC the state TRUE,
	            //means there is a parcel on sensor and Caljan runs to rising edge of BufferPEC and 300MS longer

	            #qUDT_CaljanSend.BufferPEC := NOT #iUDT_CaljanReceive.PECUnloader;

	        END_IF;

	    END_REGION


	END_REGION

	REGION 10 - Reverse run

	    IF #ix_CaljanMode = 2 THEN

	        #qUDT_CaljanSend.JogReverseCommand := #ix_ExternalRunReverse;

	    END_IF;

	END_REGION

	REGION 11 - Reset

	    // Safety ok extended pulse
	    #R_TRIG_SafetyOk(CLK := #ix_SafetyReset);

	    #s_FB_ResetPulseTimer(iudi_OffDelayTime := #iUDT_CaljanConfiguration.ResetDelay,
	                          ix_SignalToDelay := #R_TRIG_SafetyOk.Q);

	    // Send reset signal to Caljan
	    #qUDT_CaljanSend.Reset := #ix_SafetyReset OR #iqUDT_EquipmentControl.Command.Reset OR #s_FB_ResetPulseTimer.qx_DelayedSignal;

	END_REGION

	REGION 12 - Status

	    //Status
	    #s_UDT_HMIStatus.Specific.StoreMode := #iUDT_CaljanReceive.StoreModeActivated;
	    #s_UDT_HMIStatus.Specific.RunMode := #iUDT_CaljanReceive.RunModeActivated;
	    #s_UDT_HMIStatus.Specific.LowerOngoing := #iUDT_CaljanReceive.LowerOngoing;
	    #s_UDT_HMIStatus.Specific.RaisingOngoing := #iUDT_CaljanReceive.RaisingOngoing;
	    #s_UDT_HMIStatus.Specific.ChuteBlocked := #iUDT_CaljanReceive.ChuteBlockedActivated;

	    //Status
	    #s_UDT_CommonStatus.Stopped := NOT #sx_AutomaticActive;
	    #s_UDT_CommonStatus.Running := (#iUDT_CaljanReceive.BeltDirection_Unloading OR #iUDT_CaljanReceive.BeltDirection_Loading);
	    #s_UDT_CommonStatus.AutoON := #sx_Ready AND #sx_AutomaticActive;
	    #s_UDT_CommonStatus.Halted := #ix_ExternalRequestHold AND #s_UDT_CommonStatus.AutoON AND NOT #sx_EnergySaveActive;
	    #s_UDT_CommonStatus.Dieback := (NOT #iqUDT_HandShake.RTR OR #ix_ExternalRequestDieBack) AND #s_UDT_CommonStatus.AutoON AND NOT #sx_EnergySaveActive
	    AND NOT #s_UDT_CommonStatus.EnergySave AND NOT #s_UDT_CommonStatus.Running;

	    #s_UDT_CommonStatus.EnergySave := #sx_EnergySaveActive;
	    #s_UDT_CommonStatus.SafetyStop := NOT #ix_SafetyOk;

	    // HMI status update on change
	    IF #s_UDT_CommonStatusOld <> #s_UDT_CommonStatus
	    THEN
	        // HMI status initialization
	        #s_UDT_HMIStatus.Status := 0;

	        // Running
	        IF #s_UDT_CommonStatus.Running
	        THEN
	            #s_UDT_HMIStatus.Status := "DB_HMIStatusConfiguration".Running;
	        END_IF;

	        // AutoON
	        IF #s_UDT_CommonStatus.AutoON
	        THEN
	            #s_UDT_HMIStatus.Status := "DB_HMIStatusConfiguration".AutoON;
	        END_IF;

	        // Stopped
	        IF #s_UDT_CommonStatus.Stopped
	        THEN
	            #s_UDT_HMIStatus.Status := "DB_HMIStatusConfiguration".Stopped;
	        END_IF;

	        // Energy save
	        IF #s_UDT_CommonStatus.EnergySave
	        THEN
	            #s_UDT_HMIStatus.Status := "DB_HMIStatusConfiguration".EnergySave;
	        END_IF;

	        // Dieback
	        IF #s_UDT_CommonStatus.Dieback
	        THEN
	            #s_UDT_HMIStatus.Status := "DB_HMIStatusConfiguration".Dieback;
	        END_IF;

	        // Halted
	        IF #s_UDT_CommonStatus.Halted
	        THEN
	            #s_UDT_HMIStatus.Status := "DB_HMIStatusConfiguration".Halted;
	        END_IF;

	        //  PEC error
	        IF #s_UDT_HMIStatus.Specific.PEC_EoS.Jam
	        THEN
	            #s_UDT_HMIStatus.Status := "DB_HMIStatusConfiguration".PECJam;
	        END_IF;

	        // Not healthy
	        IF #s_UDT_HMIStatus.Specific.NotHealthy
	        THEN
	            #s_UDT_HMIStatus.Status := "DB_HMIStatusConfiguration".VFDNotHealthy;
	        END_IF;

	        // Safety stop
	        IF #s_UDT_CommonStatus.SafetyStop
	        THEN
	            #s_UDT_HMIStatus.Status := "DB_HMIStatusConfiguration".SafetyStop;
	        END_IF;

	        // Copy statuses

	        #s_UDT_CommonStatusOld := #s_UDT_CommonStatus;
	        #qUDT_Status := #s_UDT_CommonStatus;
	    END_IF;

	    #qUDT_HMIStatus := #s_UDT_HMIStatus;

	END_REGION

	REGION 13 - Statistics

	    // Up time
	    IF #sx_AutomaticActive
	        AND #sx_Ready
	        OR #iqUDT_EquipmentControl.Command.ResetData
	    THEN
	        "FC_Statistics"(ix_Reset := #iqUDT_EquipmentControl.Command.ResetData,
	                        ix_Activate := #sx_AutomaticActive AND #sx_Ready,
	                        ix_RTrigActivate := #R_TRIG_ConveyorUp.Q,
	                        iqUDT_Statistics := #iqUDT_Statistics.ExtendableUpTime);
	    END_IF;

	    // Down time
	    IF NOT #sx_AutomaticActive
	        AND #sx_Ready
	        OR #iqUDT_EquipmentControl.Command.ResetData
	    THEN
	        "FC_Statistics"(ix_Reset := #iqUDT_EquipmentControl.Command.ResetData,
	                        ix_Activate := NOT #sx_AutomaticActive AND #sx_Ready,
	                        ix_RTrigActivate := #R_TRIG_ConveyorDown.Q,
	                        iqUDT_Statistics := #iqUDT_Statistics.ExtendableDownTime);
	    END_IF;

	    // Energy save mode active
	    IF #sx_EnergySaveActive
	        OR #iqUDT_EquipmentControl.Command.ResetData
	    THEN
	        "FC_Statistics"(ix_Reset := #iqUDT_EquipmentControl.Command.ResetData,
	                        ix_Activate := #s_UDT_CommonStatus.EnergySave,
	                        ix_RTrigActivate := #R_TRIG_EnergySave.Q,
	                        iqUDT_Statistics := #iqUDT_Statistics.EnergySave);
	    END_IF;

	    // Not healthy
	    IF #s_UDT_HMIStatus.Specific.NotHealthy
	        OR #iqUDT_EquipmentControl.Command.ResetData
	    THEN
	        "FC_Statistics"(ix_Reset := #iqUDT_EquipmentControl.Command.ResetData,
	                        ix_Activate := #s_UDT_HMIStatus.Specific.NotHealthy,
	                        ix_RTrigActivate := #R_TRIG_NotHealthy.Q,
	                        iqUDT_Statistics := #iqUDT_Statistics.NotHealthy);
	    END_IF;

	    // PN Slave not online
	    IF #iqUDT_EquipmentControl.Command.ResetData OR #s_UDT_HMIStatus.Specific.PNSlaveNotOnline
	    THEN

	        "FC_Statistics"(ix_Reset := #iqUDT_EquipmentControl.Command.ResetData,
	                        ix_Activate := #s_UDT_HMIStatus.Specific.PNSlaveNotOnline,
	                        ix_RTrigActivate := #s_R_TRIG_PNSlaveNotOnline.Q,
	                        iqUDT_Statistics := #iqUDT_Statistics.PNNodeNotOnline);
	    END_IF;

	    // PN Slave error
	    IF #iqUDT_EquipmentControl.Command.ResetData OR #s_UDT_HMIStatus.Specific.PNSlaveError
	    THEN

	        "FC_Statistics"(ix_Reset := #iqUDT_EquipmentControl.Command.ResetData,
	                        ix_Activate := #s_UDT_HMIStatus.Specific.PNSlaveError,
	                        ix_RTrigActivate := #s_R_TRIG_PNSlaveError.Q,
	                        iqUDT_Statistics := #iqUDT_Statistics.PNNodeError);
	    END_IF;

	END_REGION

	REGION 14 - Report to control block

	    "FC_EquipmentReport"(iUDT_Status := #s_UDT_CommonStatus,
	                         iqUDT_Control := #iqUDT_EquipmentControl);

	END_REGION
END_FUNCTION_BLOCK

FUNCTION_BLOCK "FB_PNNode"
{ S7_Optimized_Access := 'TRUE' }
VERSION : 0.1
// ATTRIBUTES
// AUTO_NUMBER = True
// BLOCK_NUMBER = 224
// END_ATTRIBUTES
   VAR_INPUT
      is_PNNodeDeviceName { ExternalAccessible := 'False'; ExternalVisible := 'False'; ExternalWritable := 'False'} : String;   //   Name of the slave device
      ix_24VOk { ExternalAccessible := 'False'; ExternalVisible := 'False'; ExternalWritable := 'False'} : Bool;   //   TRUE when 24VDC is healthy
      ix_SimulationModeActive { ExternalAccessible := 'False'; ExternalVisible := 'False'; ExternalWritable := 'False'} : Bool;   //   TRUE when simulation mode active
      ix_HardwareOk { ExternalAccessible := 'False'; ExternalVisible := 'False'; ExternalWritable := 'False'} : Bool;   //  TRUE when  hardware is Ok
   END_VAR

   VAR_OUTPUT
      qUDT_HMIStatus { ExternalAccessible := 'False'; ExternalVisible := 'False'; ExternalWritable := 'False'} : "UDT_PNNodeStatus";   //   HMI status structure
      qUDT_Status { ExternalAccessible := 'False'; ExternalVisible := 'False'; ExternalWritable := 'False'} : "UDT_CommonStatus";   //   Common status structure
   END_VAR

   VAR_IN_OUT
      iqUDT_EquipmentControl : "UDT_EquipmentControl";   //   Equipment control structure
      iqUDT_Statistics : "UDT_PNNodeStatistics";   //   Statistics structure
   END_VAR

   VAR
      sUDT_CommonStatus { ExternalAccessible := 'False'; ExternalVisible := 'False'; ExternalWritable := 'False'; S7_SetPoint := 'False'} : "UDT_CommonStatus";   //   Common status structure
      sUDT_CommonStatusOld { ExternalAccessible := 'False'; ExternalVisible := 'False'; ExternalWritable := 'False'; S7_SetPoint := 'False'} : "UDT_CommonStatus";   //   Common status structure
      sUDT_HMIStatus { ExternalAccessible := 'False'; ExternalVisible := 'False'; ExternalWritable := 'False'; S7_SetPoint := 'False'} : "UDT_PNNodeStatus";   //   HMI status structure
      s_DT_PNDevice { ExternalAccessible := 'False'; ExternalVisible := 'False'; ExternalWritable := 'False'; S7_SetPoint := 'False'} : "UDT_PNDevice";   //   PN device info structure
      sa_PNPortsStatus { ExternalAccessible := 'False'; ExternalVisible := 'False'; ExternalWritable := 'False'} : Array[1..8] of Bool;   // TRUE when specific port has an error
      sFB_TimerOnOffDelayCheckSupply { ExternalAccessible := 'False'; ExternalVisible := 'False'; ExternalWritable := 'False'; S7_SetPoint := 'False'} : "FB_TimerOnOffDelay";   //   MHS "TimerOnOffDelay" - to delay time for VFD supply contactor
      sR_TRIG_PNSlaveNotOnline {InstructionName := 'R_TRIG'; LibVersion := '1.0'; ExternalAccessible := 'False'; ExternalVisible := 'False'; ExternalWritable := 'False'; S7_SetPoint := 'False'} : R_TRIG;   //   Rising edge for trigger Profinet slave not online statistics
      sR_TRIG_PNSlaveError {InstructionName := 'R_TRIG'; LibVersion := '1.0'; ExternalAccessible := 'False'; ExternalVisible := 'False'; ExternalWritable := 'False'; S7_SetPoint := 'False'} : R_TRIG;   //   Rising edge for trigger Profinet slave error statistics
      sx_PowerOk { ExternalAccessible := 'False'; ExternalVisible := 'False'; ExternalWritable := 'False'} : Bool;   //   True = External Power OK
   END_VAR

   VAR CONSTANT
      ci_PowerSupplyDelayTime : UInt := 4000;   //   Power supply delay time
      ci_NumberOfProfinetPorts : Int := 2;   // Number of Profinet ports in device
   END_VAR


BEGIN
	(*
	----------------------------------------------------------------------------------------

	Version history:
	Date        | Version   | Author        | Remark
	----------------------------------------------------------------------------------------
	28/01/2020  | 3.0       | M. Kurpiers   | first release MHS TIA 15.1
	21/04/2020  | 3.1       | S. Theocharis | renamed to PN Node
	09/07/2020  | 3.2       | S.Theocharis  | Bug fix in status update. Initialize static status instead output status
	03/11/2020  | 3.5       | K.Pokorski    | Profinet ports diagnostics added
	21/02/2023  | 4.0       | F.Baten       | 4.0 Release TIA 17.5
	*)
	REGION 1 - Get Device Profinet information

	    "FC_GetDevicePN"(is_PNDeviceName := #is_PNNodeDeviceName,
	                     ix_SimulationModeActive := #ix_SimulationModeActive,
	                     iqUDT_PND := #s_DT_PNDevice);


	    "FC_GetPNPortStatus"(ii_NumberOfPorts := #ci_NumberOfProfinetPorts,
	                         iUDT_DevicePNInfo := #s_DT_PNDevice,
	                         qa_PortFault => #sa_PNPortsStatus);

	END_REGION

	REGION 2 - Reset errors

	    // Reset Profinet Slave error/not online
	    IF #iqUDT_EquipmentControl.Command.Reset
	    THEN

	        #sUDT_HMIStatus.Specific.PNSlaveNotOnline := FALSE;
	        #sUDT_HMIStatus.Specific.PNSlaveError := FALSE;
	        #sUDT_HMIStatus.Specific.PNSlaveWarning := FALSE;

	    END_IF;

	END_REGION

	REGION 3 - Update PN slave device status

	    // Hardware will only be available after the delay, so the device has time for the initialisation
	    #sFB_TimerOnOffDelayCheckSupply(iudi_OnDelayTime := #ci_PowerSupplyDelayTime,
	                                    ix_SignalToDelay := #ix_24VOk,
	                                    qx_DelayedSignal => #sx_PowerOk);


	    // Check if PN device is online
	    IF (NOT "DB_ProfinetDiagnostic".ProfinetNetworks[#s_DT_PNDevice.PNNetworknumber].DeviceStatus[#s_DT_PNDevice.PNDeviceNumber].DeviceState.Exist
	        OR NOT #s_DT_PNDevice.PNDeviceFound)
	        AND #sx_PowerOk
	        AND NOT #ix_SimulationModeActive
	    THEN

	        #sUDT_HMIStatus.Specific.PNSlaveNotOnline := TRUE;

	    END_IF;

	    // Check if PN ports are healthy
	    IF #sa_PNPortsStatus[1] XOR #sa_PNPortsStatus[2] THEN
	        #sUDT_HMIStatus.Specific.PNSlaveWarning := TRUE;
	    END_IF;

	    // Check if PN device has an error
	    IF "DB_ProfinetDiagnostic".ProfinetNetworks[#s_DT_PNDevice.PNNetworknumber].DeviceStatus[#s_DT_PNDevice.PNDeviceNumber].DeviceState.Error
	        AND #sx_PowerOk
	        AND NOT #ix_SimulationModeActive
	        AND NOT #sUDT_HMIStatus.Specific.PNSlaveWarning
	    THEN

	        #sUDT_HMIStatus.Specific.PNSlaveError := TRUE;

	    END_IF;

	END_REGION

	REGION 4 - Statistics

	    // Create trigger on error and create statistics for profinet slave not online
	    #sR_TRIG_PNSlaveNotOnline(CLK := #sUDT_HMIStatus.Specific.PNSlaveNotOnline);

	    IF #iqUDT_EquipmentControl.Command.ResetData OR #sUDT_HMIStatus.Specific.PNSlaveNotOnline
	    THEN

	        "FC_Statistics"(ix_Reset := #iqUDT_EquipmentControl.Command.ResetData,
	                        ix_Activate := #sUDT_HMIStatus.Specific.PNSlaveNotOnline,
	                        ix_RTrigActivate := #sR_TRIG_PNSlaveNotOnline.Q,
	                        iqUDT_Statistics := #iqUDT_Statistics.PNSlaveNotOnline);

	    END_IF;

	    // Create trigger on error and create statistics for profinet slave error
	    #sR_TRIG_PNSlaveError(CLK := #sUDT_HMIStatus.Specific.PNSlaveError);

	    IF #iqUDT_EquipmentControl.Command.ResetData OR #sUDT_HMIStatus.Specific.PNSlaveError
	    THEN

	        "FC_Statistics"(ix_Reset := #iqUDT_EquipmentControl.Command.ResetData,
	                        ix_Activate := #sUDT_HMIStatus.Specific.PNSlaveError,
	                        ix_RTrigActivate := #sR_TRIG_PNSlaveError.Q,
	                        iqUDT_Statistics := #iqUDT_Statistics.PNSlaveError);

	    END_IF;

	END_REGION

	REGION 5 - Status

	    #sUDT_CommonStatus.Error := #sUDT_HMIStatus.Specific.PNSlaveError
	    OR #sUDT_HMIStatus.Specific.PNSlaveNotOnline;


	    // HMI status update
	    IF #sUDT_CommonStatusOld <> #sUDT_CommonStatus                    // update on change
	    THEN

	        // HMI status initialization
	        #sUDT_HMIStatus.Status := 0;

	        // HMI status calculation
	        IF #sUDT_HMIStatus.Specific.PNSlaveError                       // Profinet error
	            OR #sUDT_HMIStatus.Specific.PNSlaveNotOnline
	        THEN

	            #sUDT_HMIStatus.Status := "DB_HMIStatusConfiguration".ProfinetError;

	        END_IF;

	        #sUDT_CommonStatusOld := #sUDT_CommonStatus;                 // Copy status to memory
	        #qUDT_Status := #sUDT_CommonStatus;                          // Copy status to output

	    END_IF;

	    #qUDT_HMIStatus := #sUDT_HMIStatus;                          // Copy HMI status to output

	END_REGION

	REGION 6 - Report to control block

	    // Function to manage report between control block and conveyor block
	    "FC_EquipmentReport"(iUDT_Status := #sUDT_CommonStatus,
	                         iqUDT_Control := #iqUDT_EquipmentControl);

	END_REGION
END_FUNCTION_BLOCK

FUNCTION_BLOCK "FB_PneumaticBrakeUnit"
TITLE = FB_PneumaticBrakeUnit
{ S7_Optimized_Access := 'TRUE' }
AUTHOR : 'F.Baten'
VERSION : 0.1
// ATTRIBUTES
// AUTO_NUMBER = True
// BLOCK_NUMBER = 223
// END_ATTRIBUTES
//Function to control a pneumatic brake contol
   VAR_INPUT
      iUDT_PneumaticBreakConfiguration { ExternalAccessible := 'False'; ExternalVisible := 'False'; ExternalWritable := 'False'} : "UDT_PneumaticBrakeConfiguration";   // Pneumatic brake configuration structure
      ix_PECBrake { ExternalAccessible := 'False'; ExternalVisible := 'False'; ExternalWritable := 'False'} : Bool;   // TRUE when the brake photoye is not blocked
      ix_PECStop { ExternalAccessible := 'False'; ExternalVisible := 'False'; ExternalWritable := 'False'} : Bool;   // TRUE when the stop photoye is not blocked
      ix_PECdownstream { ExternalAccessible := 'False'; ExternalVisible := 'False'; ExternalWritable := 'False'} : Bool;   // TRUE when the photoye downstream is not blocked
      ix_DownstreamStopActive { ExternalAccessible := 'False'; ExternalVisible := 'False'; ExternalWritable := 'False'} : Bool;   // TRUE when the downstream stop is active
      ix_MasterValve { ExternalAccessible := 'False'; ExternalVisible := 'False'; ExternalWritable := 'False'} : Bool;   // TRUE when master valve is on
      ix_SafetyOk { ExternalAccessible := 'False'; ExternalVisible := 'False'; ExternalWritable := 'False'} : Bool;   // TRUE when safety is ok
   END_VAR

   VAR_OUTPUT
      qx_Valve { ExternalAccessible := 'False'; ExternalVisible := 'False'; ExternalWritable := 'False'} : Bool;   // TRUE when valve is activated
      qx_StopActive { ExternalAccessible := 'False'; ExternalVisible := 'False'; ExternalWritable := 'False'} : Bool;   // TRUE when stop is activated to upstream
   END_VAR

   VAR_IN_OUT
      iqUDT_EquipmentControl : "UDT_EquipmentControl";   // Equipment control structure
   END_VAR

   VAR
      s_PECBreakTimerOnOffDelay { ExternalAccessible := 'False'; ExternalVisible := 'False'; ExternalWritable := 'False'; S7_SetPoint := 'False'} : "FB_TimerOnOffDelay";   // Filtering end of section photo eye signal
      s_PECStopTimerOnOffDelay { ExternalAccessible := 'False'; ExternalVisible := 'False'; ExternalWritable := 'False'; S7_SetPoint := 'False'} : "FB_TimerOnOffDelay";   // Filtering end of section photo eye signal
      s_StopFunctionTimerOnOffDelay { ExternalAccessible := 'False'; ExternalVisible := 'False'; ExternalWritable := 'False'; S7_SetPoint := 'False'} : "FB_TimerOnOffDelay";   // Filtering end of section photo eye signal
      s_StopReleaseOnOffDelay { ExternalAccessible := 'False'; ExternalVisible := 'False'; ExternalWritable := 'False'; S7_SetPoint := 'False'} : "FB_TimerOnOffDelay";
      sR_TRIG_PECStop {InstructionName := 'R_TRIG'; LibVersion := '1.0'; ExternalAccessible := 'False'; ExternalVisible := 'False'; ExternalWritable := 'False'; S7_SetPoint := 'False'} : R_TRIG;   // Rising edge trigger PEC jam
      slr_StepTimer { ExternalAccessible := 'False'; ExternalVisible := 'False'; ExternalWritable := 'False'} : LReal;   // Step timer
      slr_BrakeInterval { ExternalAccessible := 'False'; ExternalVisible := 'False'; ExternalWritable := 'False'} : LReal;   // Brake interval
      si_BrakeFunction { ExternalAccessible := 'False'; ExternalVisible := 'False'; ExternalWritable := 'False'} : Int;   // Brake function step
      si_BrakeCycles { ExternalAccessible := 'False'; ExternalVisible := 'False'; ExternalWritable := 'False'} : Int;   // Number of cyles
      sx_Cycle { ExternalAccessible := 'False'; ExternalVisible := 'False'; ExternalWritable := 'False'} : Bool;   // Cycle
      sx_PECBrakeFiltered { ExternalAccessible := 'False'; ExternalVisible := 'False'; ExternalWritable := 'False'} : Bool;   // PEC signal filtered
      sx_PECStopFiltered { ExternalAccessible := 'False'; ExternalVisible := 'False'; ExternalWritable := 'False'} : Bool;   // PEC signal filtered
      sx_DownstreamStop { ExternalAccessible := 'False'; ExternalVisible := 'False'; ExternalWritable := 'False'} : Bool;   // Downstream is stopped
      sx_StopFunctionActive { ExternalAccessible := 'False'; ExternalVisible := 'False'; ExternalWritable := 'False'} : Bool;   // Stop function is activated
      sx_BrakePulse { ExternalAccessible := 'False'; ExternalVisible := 'False'; ExternalWritable := 'False'} : Bool;   // Brake pulse 1 is active
      sx_BrakeAssemblyValve { ExternalAccessible := 'False'; ExternalVisible := 'False'; ExternalWritable := 'False'} : Bool;   // Brake assembly valve
      sx_NoCycles { ExternalAccessible := 'False'; ExternalVisible := 'False'; ExternalWritable := 'False'} : Bool;   // No cycles
      sx_Enable_release { ExternalAccessible := 'False'; ExternalVisible := 'False'; ExternalWritable := 'False'} : Bool;
   END_VAR

   VAR CONSTANT
      ci_ReleaseStopBreakTimeOnDelay : UInt := 10000;
   END_VAR


BEGIN
	(*
	----------------------------------------------------------------------------------------

	Version history:
	Date        | Version   | Author        | Remark
	----------------------------------------------------------------------------------------
	23/06/2021  | 0.0       | F. Baten      | first release TIA 15.1
	20/10/2021  | 0.1       | M. Piela      | Add equipment control. Stylistic correction
	25/06/2021  | 0.2       | M. Kurpiers   | Add stop break release
	21/02/2023  | 4.0       | F.Baten       | 4.0 Release TIA 17.5
	 *)

	REGION 1 - Timers

	    // Filtering brake photo eye signal
	    #s_PECBreakTimerOnOffDelay(iudi_OnDelayTime := #iUDT_PneumaticBreakConfiguration.PECBrakeOnDelay,
	                               iudi_OffDelayTime := #iUDT_PneumaticBreakConfiguration.PECBrakeOffDelay,
	                               ix_SignalToDelay := #ix_PECBrake,
	                               ix_Enable := TRUE,
	                               qx_DelayedSignal => #sx_PECBrakeFiltered);

	    // Filtering stop photo eye signal
	    #s_PECStopTimerOnOffDelay(iudi_OnDelayTime := #iUDT_PneumaticBreakConfiguration.PECStopOnDelay,
	                              iudi_OffDelayTime := #iUDT_PneumaticBreakConfiguration.PECStopOffDelay,
	                              ix_SignalToDelay := #ix_PECStop,
	                              ix_Enable := TRUE,
	                              qx_DelayedSignal => #sx_PECStopFiltered);

	    // Filtering downstream stop photo eye signal
	    #s_StopFunctionTimerOnOffDelay(iudi_OnDelayTime := #iUDT_PneumaticBreakConfiguration.StopFunctionOnDelay,
	                                   iudi_OffDelayTime := #iUDT_PneumaticBreakConfiguration.StopFunctionOffDelay,
	                                   ix_SignalToDelay := #ix_DownstreamStopActive,
	                                   ix_Enable := TRUE,
	                                   qx_DelayedSignal => #sx_DownstreamStop);

	    #s_StopReleaseOnOffDelay(iudi_OnDelayTime := #ci_ReleaseStopBreakTimeOnDelay,
	                             iudi_OffDelayTime := 0,
	                             ix_SignalToDelay := #ix_PECdownstream AND NOT #ix_PECBrake,
	                             ix_Enable := TRUE,
	                             qx_DelayedSignal => #sx_Enable_release);

	    // Sequence Timer
	    IF #slr_StepTimer > 0
	    THEN
	        #slr_StepTimer -= "DB_Memory".PrevCycleTime;
	        IF #slr_StepTimer < 0
	        THEN
	            #slr_StepTimer := 0;
	        END_IF;
	    END_IF;

	END_REGION

	REGION 2 - Brake function
	    // Braking of the parcel is activated when first parcel arrives in brake PEC and stop function is not active.
	    // Now the brake is raised configured number of times with the configured brakepuls time and the configured delay. this is done every time again with the configured
	    // interval time as long as the PEC brake is occupied.

	    #sR_TRIG_PECStop(CLK := #ix_PECStop);
	    // Restart sequence
	    IF #sR_TRIG_PECStop.Q AND NOT #sx_PECStopFiltered
	    THEN
	        #si_BrakeFunction := 1;
	    END_IF;

	    IF #sx_NoCycles AND #ix_PECBrake THEN
	        #sx_NoCycles := FALSE;
	    END_IF;

	    IF #iUDT_PneumaticBreakConfiguration.BrakeCycles = 1
	    THEN
	        #slr_BrakeInterval := #iUDT_PneumaticBreakConfiguration.BrakePause;
	    ELSE
	        #slr_BrakeInterval := #iUDT_PneumaticBreakConfiguration.BrakeInterval;
	    END_IF;
	    // Sequence
	    IF #si_BrakeFunction = 1 AND #slr_StepTimer = 0 AND (NOT #ix_PECBrake OR #sx_BrakePulse)
	    THEN
	        #sx_BrakePulse := TRUE;
	        #slr_StepTimer := #iUDT_PneumaticBreakConfiguration.BrakePuls;
	        #si_BrakeFunction := 2;
	        #sx_Cycle := TRUE;
	    END_IF;

	    IF (#si_BrakeFunction = 2 OR #sx_Enable_release) AND #slr_StepTimer = 0 AND #ix_SafetyOk
	    THEN
	        #sx_BrakePulse := False;
	        #si_BrakeCycles += 1;
	        IF #iUDT_PneumaticBreakConfiguration.BrakeCycles > 0
	        THEN
	            IF #si_BrakeCycles >= #iUDT_PneumaticBreakConfiguration.BrakeCycles
	            THEN
	                #si_BrakeCycles := 0;
	                #slr_StepTimer := #slr_BrakeInterval;
	                #si_BrakeFunction := 3;
	                #sx_Cycle := TRUE;
	            ELSE
	                #slr_StepTimer := #iUDT_PneumaticBreakConfiguration.BrakePause;
	                #si_BrakeFunction := 1;
	                #sx_Cycle := TRUE;
	            END_IF;
	        ELSE
	            #sx_NoCycles := TRUE;
	            #si_BrakeCycles := 0;
	            #si_BrakeFunction := 4;
	        END_IF;
	    END_IF;
	    // Waiting time between interval
	    IF (#si_BrakeFunction = 3 AND #slr_StepTimer = 0) OR #sx_StopFunctionActive
	    THEN
	        #si_BrakeFunction := 1;
	    END_IF;
	    // Wait for pec to clear, one puls only
	    IF (#si_BrakeFunction = 4 AND NOT #sx_NoCycles) OR #sx_StopFunctionActive
	    THEN
	        #si_BrakeFunction := 1;
	    END_IF;

	END_REGION

	REGION 3 - Brake valve

	    REGION 3.1 - Brake assembly valve function

	        IF #sx_StopFunctionActive AND NOT #sx_DownstreamStop
	        THEN
	            #sx_StopFunctionActive := FALSE;
	        END_IF;

	        IF #sx_DownstreamStop AND NOT #sx_PECStopFiltered AND NOT #sx_PECBrakeFiltered
	        THEN
	            #sx_StopFunctionActive := TRUE;
	        END_IF;

	        #sx_BrakeAssemblyValve := (#sx_StopFunctionActive
	        AND ((#iUDT_PneumaticBreakConfiguration.Slave AND #ix_MasterValve)
	        OR NOT #iUDT_PneumaticBreakConfiguration.Slave))
	        OR (NOT #sx_StopFunctionActive
	        AND #sx_BrakePulse);

	    END_REGION

	    REGION 3.2 Valve activation

	        IF #iUDT_PneumaticBreakConfiguration.FailSafe
	        THEN
	            #qx_Valve := NOT (#sx_BrakeAssemblyValve OR NOT #ix_SafetyOk);
	        ELSE
	            #qx_Valve := #sx_BrakeAssemblyValve AND #ix_SafetyOk;
	        END_IF;

	    END_REGION

	END_REGION

	REGION 4 - Stop Active

	    #qx_StopActive := #sx_StopFunctionActive AND NOT #sx_PECStopFiltered AND NOT #sx_PECBrakeFiltered;

	END_REGION
END_FUNCTION_BLOCK

FUNCTION_BLOCK "FB_Capacity"
{ S7_Optimized_Access := 'TRUE' }
VERSION : 0.1
// ATTRIBUTES
// AUTO_NUMBER = True
// BLOCK_NUMBER = 202
// END_ATTRIBUTES
   VAR_INPUT
      iUDT_CapacityConfiguration { ExternalAccessible := 'False'; ExternalVisible := 'False'; ExternalWritable := 'False'} : "UDT_CapacityConfiguration";   // Capacity configuration structure
      ix_PECFiltered { ExternalAccessible := 'False'; ExternalVisible := 'False'; ExternalWritable := 'False'} : Bool;   // TRUE when the end of section photoeye is not blocked
      ix_ResetData { ExternalAccessible := 'False'; ExternalVisible := 'False'; ExternalWritable := 'False'} : Bool;   // Reset data
   END_VAR

   VAR_OUTPUT
      qx_Error { ExternalAccessible := 'False'; ExternalVisible := 'False'; ExternalWritable := 'False'} : Bool;   // TRUE when collective block error occurred
      qx_Warning { ExternalAccessible := 'False'; ExternalVisible := 'False'; ExternalWritable := 'False'} : Bool;   // TRUE when collective block warning occurred
      qi_Capacity { ExternalAccessible := 'False'; ExternalVisible := 'False'; ExternalWritable := 'False'} : Int;   // Capacity value
      qa_CapacityBuffer { ExternalAccessible := 'False'; ExternalVisible := 'False'; ExternalWritable := 'False'} : Array[0..#Samples] of Int;   // Capacity buffer
      qa_PPHBuffer { ExternalAccessible := 'False'; ExternalVisible := 'False'; ExternalWritable := 'False'} : Array[0..#Samples] of Int;   // Parcel per hour buffer
   END_VAR

   VAR_IN_OUT
      iqUDT_ConveyorInterface : "UDT_ConveyorInterface";   // Conveyor interface
   END_VAR

   VAR
      sFB_Pulse { ExternalAccessible := 'False'; ExternalVisible := 'False'; ExternalWritable := 'False'; S7_SetPoint := 'False'} : "FB_Pulse";   // Function block to generate custom pulse signal.
      sR_TRIG_ParcelDetect {InstructionName := 'R_TRIG'; LibVersion := '1.0'; ExternalAccessible := 'False'; ExternalVisible := 'False'; ExternalWritable := 'False'; S7_SetPoint := 'False'} : R_TRIG;   // Parcel detect
      sa_Status { ExternalAccessible := 'False'; ExternalVisible := 'False'; ExternalWritable := 'False'} : Struct   // Status structure
         FifoError { ExternalAccessible := 'False'; ExternalVisible := 'False'; ExternalWritable := 'False'} : Bool;   //    FIFO block error
         FifoWarning { ExternalAccessible := 'False'; ExternalVisible := 'False'; ExternalWritable := 'False'} : Bool;   //    FIFO block warning
         ConfigurationError { ExternalAccessible := 'False'; ExternalVisible := 'False'; ExternalWritable := 'False'} : Bool;   //    Collective configuration error
      END_STRUCT;
      sr_CollectiveParcelLength { ExternalAccessible := 'False'; ExternalVisible := 'False'; ExternalWritable := 'False'} : Real;   // Colletive parcel length [mm]
      sr_ParcelCount { ExternalAccessible := 'False'; ExternalVisible := 'False'; ExternalWritable := 'False'} : Real;   // Parcel count
      sr_RecalculatedWindow { ExternalAccessible := 'False'; ExternalVisible := 'False'; ExternalWritable := 'False'} : Real;   // Window recalculated based on configured avg parcel length
      sr_ParcelPerHour { ExternalAccessible := 'False'; ExternalVisible := 'False'; ExternalWritable := 'False'} : Real;   // Parcel(s) per hour
      sr_AveragePackageLength { ExternalAccessible := 'False'; ExternalVisible := 'False'; ExternalWritable := 'False'} : Real;   // Average parcel length [mm]
      sr_AverageGap { ExternalAccessible := 'False'; ExternalVisible := 'False'; ExternalWritable := 'False'} : Real;   // Average gap size [mm]
      sr_AverageWindow { ExternalAccessible := 'False'; ExternalVisible := 'False'; ExternalWritable := 'False'} : Real;   // Average window size [mm]
      sudi_Interval { ExternalAccessible := 'False'; ExternalVisible := 'False'; ExternalWritable := 'False'} : UDInt;   // Interval [ms]
      si_Capacity { ExternalAccessible := 'False'; ExternalVisible := 'False'; ExternalWritable := 'False'} : Int;   // Capacity value for the configured package length
      si_ConveyorDistanceTraveled { ExternalAccessible := 'False'; ExternalVisible := 'False'; ExternalWritable := 'False'} : Int;   // Distance the conveyour travelled this interval
      sx_ParcelDetected { ExternalAccessible := 'False'; ExternalVisible := 'False'; ExternalWritable := 'False'} : Bool := FALSE;   // Parcel detected
      sx_SendData { ExternalAccessible := 'False'; ExternalVisible := 'False'; ExternalWritable := 'False'} : Bool;   // Send data signal
   END_VAR

   VAR CONSTANT
      Samples : ULInt := 120;
   END_VAR


BEGIN
	(*
	----------------------------------------------------------------------------------------

	Version history:
	Date        | Version   | Author        | Remark
	----------------------------------------------------------------------------------------
	21/01/2020  | 3.0       | A.Nowak       | Initial version
	14/02/2020  | 3.1       | A.Nowak       | Add sample amount and treshold to the configuration and reset data functionality
	13/03/2020  | 3.2       | M.Kurpiers    | Adapting reviews
	23/03/2020  | 3.3       | A. Nowak      | Change the values to the mm
	20/04/2022  | 3.4       | M.Roijen      | Remove MFC logging and added the shift of data
	06/08/2022  | 3.5       | M.Singh       | add Reset PPH Buffer and used avg Length from Config.
	15/05/2023  | 4.0       | F.Baten       | 4.0 Release TIA 17.5
	                                          Removed 'si_DataCounter', 'si_Displacement', 'iUDT_CapacityConfiguration.SampleAmount', fixed 'sr_AveragePackageLength' calculation
	                                          Added constant 'Samples' for length of arrays.
	*)

	REGION 1 - Configuration check

	    // If the block is configured properly, convert interval to the ms and reset the error. Otherwise, set configuration error.
	    IF #iUDT_CapacityConfiguration.Interval > 0
	        AND #iUDT_CapacityConfiguration.AveragePackageLengthConfiguration > 0
	        AND #iUDT_CapacityConfiguration.Treshold >= 0
	    THEN
	        #sudi_Interval := #iUDT_CapacityConfiguration.Interval * 1000;
	        #sa_Status.ConfigurationError := FALSE;
	    ELSE
	        #sa_Status.ConfigurationError := TRUE;
	    END_IF;

	END_REGION

	REGION 2 - Reset data

	    // If there is reset data request, initialize sample amount and data buffer.
	    IF #ix_ResetData
	    THEN
	        FILL_BLK(IN := 0,
	                 COUNT := #Samples,
	                 OUT => #qa_CapacityBuffer[0]);
	        FILL_BLK(IN := 0,
	                 COUNT := #Samples,
	                 OUT => #qa_PPHBuffer[0]);
	    END_IF;

	END_REGION

	REGION 4 - PEC

	    #sx_ParcelDetected := NOT #ix_PECFiltered;

	END_REGION

	REGION 5 - Interval check

	    // Generate puls signal every interval.
	    #sFB_Pulse(iudi_PulseTime := #sudi_Interval,
	               qx_Pulse => #sx_SendData);

	END_REGION

	REGION 6 - Package length measurement and parcel count

	    // Parcel is detected.
	    IF #sx_ParcelDetected
	    THEN
	        // Add displacement to the collective parcel length.
	        #sr_CollectiveParcelLength += (ABS(#iqUDT_ConveyorInterface.Displacement)) * 10;
	    END_IF;

	    #sR_TRIG_ParcelDetect(CLK := #sx_ParcelDetected);
	    // Increment parcel count when package is detected.
	    IF #sR_TRIG_ParcelDetect.Q
	    THEN
	        #sr_ParcelCount += 1;
	    END_IF;

	    // Measure the distance traveled by conveyor
	    #si_ConveyorDistanceTraveled += (ABS(#iqUDT_ConveyorInterface.Displacement)) * 10;

	END_REGION

	REGION 7 - Capacity calculation and data send

	    // There is no configuration error and there are send data and enable signals.
	    IF NOT #sa_Status.ConfigurationError
	        AND #sx_SendData
	    THEN
	        // Parcel was detected.
	        IF #sr_ParcelCount <> 0
	            AND #sr_CollectiveParcelLength <> 0
	        THEN
	            // Calculate average values.
	            #sr_AveragePackageLength := #sr_CollectiveParcelLength / #sr_ParcelCount;
	            #sr_AverageWindow := #si_ConveyorDistanceTraveled / #sr_ParcelCount;
	            #sr_AverageGap := #sr_AverageWindow - #sr_AveragePackageLength;

	            // Windowsize calculated based on configured average parcel length
	            #sr_RecalculatedWindow := #sr_AverageGap + #iUDT_CapacityConfiguration.AveragePackageLengthConfiguration;

	            // Calculate parcel per hour value for the configured average parcel length.
	            #si_Capacity := DINT_TO_INT(TRUNC((#sr_ParcelPerHour * #sr_AverageWindow) / #sr_RecalculatedWindow));

	            // Calculate parcel per hour value using data from the interval.
	            #sr_ParcelPerHour := (#sr_ParcelCount / UDINT_TO_REAL(#iUDT_CapacityConfiguration.Interval)) * 3600;

	        ELSE
	            #si_Capacity := 0;
	        END_IF;

	        #qi_Capacity := #si_Capacity;

	        // Capacity value is greater than configured treshold.
	        IF #si_Capacity >= #iUDT_CapacityConfiguration.Treshold
	        THEN
	            MOVE_BLK(IN := #qa_CapacityBuffer[0],
	                     COUNT := #Samples,
	                     OUT => #qa_CapacityBuffer[1]);
	            #qa_CapacityBuffer[0] := #si_Capacity;

	            MOVE_BLK(IN := #qa_PPHBuffer[0],
	                     COUNT := #Samples,
	                     OUT => #qa_PPHBuffer[1]);
	            #qa_PPHBuffer[0] := REAL_TO_INT(#sr_ParcelPerHour);
	        END_IF;

	        // Initialize parcel count and collective parcel length.
	        #sr_ParcelCount := 0;
	        #sr_CollectiveParcelLength := 0;
	        #si_ConveyorDistanceTraveled := 0;
	    END_IF;

	END_REGION

	REGION 8 - Status

	    // Collective error.
	    #qx_Error :=
	    #sa_Status.ConfigurationError
	    OR #sa_Status.FifoError;

	    // Collective warning.
	    #qx_Warning := #sa_Status.FifoWarning;

	END_REGION
END_FUNCTION_BLOCK

FUNCTION_BLOCK "FB_Chute1PEC"
{ S7_Optimized_Access := 'TRUE' }
VERSION : 0.1
// ATTRIBUTES
// AUTO_NUMBER = True
// BLOCK_NUMBER = 203
// END_ATTRIBUTES
   VAR_INPUT
      iUDT_ChuteConfiguration { ExternalAccessible := 'False'; ExternalVisible := 'False'; ExternalWritable := 'False'} : "UDT_Chute1PECConfiguration";   // Chute Configuration structure
      iUDT_UpstreamConveyorStatus { ExternalAccessible := 'False'; ExternalVisible := 'False'; ExternalWritable := 'False'} : "UDT_CommonStatus";   // Upstream conveyor status
      ix_PECFull { ExternalAccessible := 'False'; ExternalVisible := 'False'; ExternalWritable := 'False'} : Bool;   // TRUE when Chute Full photoeye is not blocked
      ix_Disabled { ExternalAccessible := 'False'; ExternalVisible := 'False'; ExternalWritable := 'False'} : Bool;   // TRUE when chute is disabled
      ix_HardwareOk { ExternalAccessible := 'False'; ExternalVisible := 'False'; ExternalWritable := 'False'} : Bool;   // TRUE when chute hardware is Ok
      iudi_DelayHardwareOK { ExternalAccessible := 'False'; ExternalVisible := 'False'; ExternalWritable := 'False'} : UDInt;   // Time to delay for hardware ok signal
   END_VAR

   VAR_OUTPUT
      qx_Lamp { ExternalAccessible := 'False'; ExternalVisible := 'False'; ExternalWritable := 'False'} : Bool;   // Output Chute Lamp full
      qUDT_HMIStatus { ExternalAccessible := 'False'; ExternalVisible := 'False'; ExternalWritable := 'False'} : "UDT_Chute1PECStatus";   // HMI status structure
      qUDT_Status { ExternalAccessible := 'False'; ExternalVisible := 'False'; ExternalWritable := 'False'} : "UDT_CommonStatus";   // Common status structure
   END_VAR

   VAR_IN_OUT
      iqUDT_EquipmentControl : "UDT_EquipmentControl";   // Equipment control structure
      iqUDT_UpstreamConveyorHandshake : "UDT_ConveyorHandshake";   // Upstream handshake structure
      iqUDT_Statistics : "UDT_Chute1PECStatistics";   // Statistics structure
   END_VAR

   VAR
      s_UDT_CommonStatus { ExternalAccessible := 'False'; ExternalVisible := 'False'; ExternalWritable := 'False'; S7_SetPoint := 'False'} : "UDT_CommonStatus";   // Common status structure
      s_UDT_CommonStatus_1 { ExternalAccessible := 'False'; ExternalVisible := 'False'; ExternalWritable := 'False'; S7_SetPoint := 'False'} : "UDT_CommonStatus";
      s_UDT_CommonStatus_2 { ExternalAccessible := 'False'; ExternalVisible := 'False'; ExternalWritable := 'False'; S7_SetPoint := 'False'} : "UDT_CommonStatus";
      s_UDT_CommonStatus_3 { ExternalAccessible := 'False'; ExternalVisible := 'False'; ExternalWritable := 'False'; S7_SetPoint := 'False'} : "UDT_CommonStatus";
      s_UDT_CommonStatus_4 { ExternalAccessible := 'False'; ExternalVisible := 'False'; ExternalWritable := 'False'; S7_SetPoint := 'False'} : "UDT_CommonStatus";
      s_UDT_CommonStatus_5 { ExternalAccessible := 'False'; ExternalVisible := 'False'; ExternalWritable := 'False'; S7_SetPoint := 'False'} : "UDT_CommonStatus";
      s_UDT_CommonStatus_6 { ExternalAccessible := 'False'; ExternalVisible := 'False'; ExternalWritable := 'False'; S7_SetPoint := 'False'} : "UDT_CommonStatus";
      s_UDT_CommonStatus_7 { ExternalAccessible := 'False'; ExternalVisible := 'False'; ExternalWritable := 'False'; S7_SetPoint := 'False'} : "UDT_CommonStatus";
      s_UDT_CommonStatus_8 { ExternalAccessible := 'False'; ExternalVisible := 'False'; ExternalWritable := 'False'; S7_SetPoint := 'False'} : "UDT_CommonStatus";
      s_UDT_CommonStatus_9 { ExternalAccessible := 'False'; ExternalVisible := 'False'; ExternalWritable := 'False'; S7_SetPoint := 'False'} : "UDT_CommonStatus";
      s_UDT_CommonStatus_10 { ExternalAccessible := 'False'; ExternalVisible := 'False'; ExternalWritable := 'False'; S7_SetPoint := 'False'} : "UDT_CommonStatus";
      s_UDT_HMIStatus { ExternalAccessible := 'False'; ExternalVisible := 'False'; ExternalWritable := 'False'; S7_SetPoint := 'False'} : "UDT_Chute1PECStatus";   // HMI status structure
      s_UDT_CommonStatusOld { ExternalAccessible := 'False'; ExternalVisible := 'False'; ExternalWritable := 'False'; S7_SetPoint := 'False'} : "UDT_CommonStatus";   // Auxiliary status structure
      s_FB_HardwareOK { ExternalAccessible := 'False'; ExternalVisible := 'False'; ExternalWritable := 'False'; S7_SetPoint := 'False'} : "FB_TimerOnOffDelay";   // Timer on/off delay for hardware ok signal
      s_FB_ChuteFullDetectionDelay { ExternalAccessible := 'False'; ExternalVisible := 'False'; ExternalWritable := 'False'; S7_SetPoint := 'False'} : "FB_TimerOnOffDelay";   // Timer on/off delay for chute full detection
      s_R_TRIG_ChuteFull {InstructionName := 'R_TRIG'; LibVersion := '1.0'; ExternalAccessible := 'False'; ExternalVisible := 'False'; ExternalWritable := 'False'; S7_SetPoint := 'False'} : R_TRIG;   // Rising edge trigger on chute full signal
      s_R_TRIG_Disabled {InstructionName := 'R_TRIG'; LibVersion := '1.0'; ExternalAccessible := 'False'; ExternalVisible := 'False'; ExternalWritable := 'False'; S7_SetPoint := 'False'} : R_TRIG;   // Rising edge trigger on chute disabled signal
      s_F_TRIG_UpdateStatus {InstructionName := 'F_TRIG'; LibVersion := '1.0'; ExternalAccessible := 'False'; ExternalVisible := 'False'; ExternalWritable := 'False'; S7_SetPoint := 'False'} : F_TRIG;   // Falling edge trigger on status change
      sx_Full { ExternalAccessible := 'False'; ExternalVisible := 'False'; ExternalWritable := 'False'} : Bool;   // Full status
   END_VAR


BEGIN
	(*
	----------------------------------------------------------------------------------------

	Version history:
	Date        | Version   | Author        | Remark
	----------------------------------------------------------------------------------------
	13/10/2021  | 0.1       | J. Krawczuk   | first release TIA 16.0
	29/10/2021  | 0.1       | M. Piela      | Design change, comments corrections
	14/01/2022  | 0.2       | G. Vlooswijk  | Fixed statistics reset
	25/07/2022  | 0.3       | M. Kurpiers   | HMI Initilization added
	30/07/2022  | 0.3       | G. Vlooswijk  | Removed running and energy save status for FedEx Scada
	21/02/2023  | 4.0       | F.Baten       | 4.0 Release TIA 17.5
	12/03/2024  | 4.1       | S. Nieswiec   | Updated variable names to current standard
	 *)

	REGION 1 - Timers

	    // Full detection timer
	    #s_FB_ChuteFullDetectionDelay(iudi_OnDelayTime := #iUDT_ChuteConfiguration.FullDetectionTime,
	                                  iudi_OffDelayTime := #iUDT_ChuteConfiguration.FullReleaseTime,
	                                  ix_SignalToDelay := NOT #ix_PECFull,
	                                  qx_DelayedSignal => #sx_Full);

	    // Hardware ok timer
	    #s_FB_HardwareOK(iudi_OnDelayTime := #iudi_DelayHardwareOK,
	                     ix_SignalToDelay := #ix_HardwareOk);

	END_REGION

	REGION 2 - Stop upstream conveyor

	    // Stop upstream conveyor when chute is full or disabled
	    #iqUDT_UpstreamConveyorHandshake.RTR := NOT #sx_Full AND NOT #ix_Disabled AND #s_FB_HardwareOK.qx_DelayedSignal;

	END_REGION

	REGION 3 - Update output

	    // Update the outputs
	    #qx_Lamp := #sx_Full;

	END_REGION

	REGION 4 - Status

	    // HMI status initialization
	    #s_UDT_HMIStatus.Status := 0;

	    // Update chute full specific status
	    #s_UDT_HMIStatus.Specific.ChuteFull := #sx_Full AND #s_FB_HardwareOK.qx_DelayedSignal;

	    //Update chute disabled specific status
	    #s_UDT_HMIStatus.Specific.ChuteDisabled := #ix_Disabled AND #s_FB_HardwareOK.qx_DelayedSignal;

	    // Update common safety stop
	    #s_UDT_CommonStatus.SafetyStop := #iUDT_UpstreamConveyorStatus.SafetyStop;

	    // Update common automatic on
	    #s_UDT_CommonStatus.AutoON := #iUDT_UpstreamConveyorStatus.AutoON;

	    // Update common stopped
	    #s_UDT_CommonStatus.Stopped := #iUDT_UpstreamConveyorStatus.Stopped;

	    // Update HMI status number for chute disabled
	    IF #s_UDT_HMIStatus.Specific.ChuteDisabled AND NOT #s_UDT_CommonStatus.SafetyStop
	    THEN
	        #s_UDT_HMIStatus.Status := "DB_HMIStatusConfiguration".DisableByManagement;

	    END_IF;

	    // Update HMI status number for chute full
	    IF #s_UDT_HMIStatus.Specific.ChuteFull AND NOT #s_UDT_CommonStatus.SafetyStop
	    THEN
	        #s_UDT_HMIStatus.Status := "DB_HMIStatusConfiguration".ChuteFull;

	    END_IF;

	    // Collecting F_TRIG on chute full or chute disabled status to update common status
	    #s_F_TRIG_UpdateStatus(CLK := #s_UDT_HMIStatus.Specific.ChuteFull OR #s_UDT_HMIStatus.Specific.ChuteDisabled);

	    // HMI status number calculation
	    IF #s_UDT_CommonStatusOld <> #s_UDT_CommonStatus OR #s_F_TRIG_UpdateStatus.Q
	    THEN

	        // Update auto on status number
	        IF #s_UDT_CommonStatus.AutoON
	        THEN
	            #s_UDT_HMIStatus.Status := "DB_HMIStatusConfiguration".AutoON;

	        END_IF;

	        IF #s_UDT_CommonStatus.Stopped
	        THEN
	            #s_UDT_HMIStatus.Status := "DB_HMIStatusConfiguration".Stopped;

	        END_IF;

	        IF #s_UDT_CommonStatus.SafetyStop
	        THEN
	            #s_UDT_HMIStatus.Status := "DB_HMIStatusConfiguration".SafetyStop;

	        END_IF;

	        // Copy common status structure to the old common status structure
	        #s_UDT_CommonStatusOld := #s_UDT_CommonStatus;
	        #qUDT_Status := #s_UDT_CommonStatus;

	    END_IF;

	    #qUDT_HMIStatus := #s_UDT_HMIStatus;


	END_REGION

	REGION 5 - Statistics

	    // Chute full R_TRIG for statistics purpose
	    #s_R_TRIG_ChuteFull(CLK := #s_UDT_HMIStatus.Specific.ChuteFull);

	    // Chute full statistics
	    IF #s_UDT_HMIStatus.Specific.ChuteFull
	        OR #iqUDT_EquipmentControl.Command.ResetData
	    THEN
	        "FC_Statistics"(ix_Reset := #iqUDT_EquipmentControl.Command.ResetData,
	                        ix_Activate := #s_UDT_HMIStatus.Specific.ChuteFull,
	                        ix_RTrigActivate := #s_R_TRIG_ChuteFull.Q,
	                        iqUDT_Statistics := #iqUDT_Statistics.ChuteFull);

	    END_IF;

	    // Chute disabled R_TRIG for statistics purpose
	    #s_R_TRIG_Disabled(CLK := #s_UDT_HMIStatus.Specific.ChuteDisabled);

	    // Chute disabled statistics
	    IF #s_UDT_HMIStatus.Specific.ChuteDisabled
	        OR #iqUDT_EquipmentControl.Command.ResetData
	    THEN
	        "FC_Statistics"(ix_Reset := #iqUDT_EquipmentControl.Command.ResetData,
	                        ix_Activate := #s_UDT_HMIStatus.Specific.ChuteDisabled,
	                        ix_RTrigActivate := #s_R_TRIG_Disabled.Q,
	                        iqUDT_Statistics := #iqUDT_Statistics.ChuteDisabled);

	    END_IF;

	END_REGION

	REGION 6 - Equipment Report

	    "FC_EquipmentReport"(iUDT_Status := #s_UDT_CommonStatus,
	                         iqUDT_Control := #iqUDT_EquipmentControl);

	END_REGION
END_FUNCTION_BLOCK

